(* CODESYS project Rasi_feeds_batching3.project

Project tree, tasks and I/O mapping:
  PLC_AC500_V3 : PM5032-T-ETH, ABB AG, order no. 1SAP123400R0x72, version 3.7.0.0
    application Application
      libraries: ModbusRtu, * (ABB); Util, * (System)
      task Task (cyclic, interval t#10ms, priority 14, watchdog t#20ms x 1) calls batching16
      CheckConfigurationObject
      Diagnosis/
        text list Diag_IO_Bus
        text list Diag_V3_PLC
      global variables GVL
      function block FB_Samyak_Multi [ST]
      function block FB_Samyak_Control [ST]
      function block Auto_Batching_V16 [ST]
      global variables PersistentVars
      function block Semi_Auto_Batching_V16 [ST]
      program batching16 [FBD]
    OnBoard_IO : 12DI/8DO-T/2DC, ABB AG, version 3.7.0.0
        input  E_Stop_DI : BOOL  // Fast inputs DI0-DI3.Digital input DI0
        input  Main_Cont_FB : BOOL  // Fast inputs DI0-DI3.Digital input DI1
        input  Auto_Mode_FB : BOOL  // Fast inputs DI0-DI3.Digital input DI2
        input  VFD_Run : BOOL  // Fast inputs DI0-DI3.Digital input DI3
        input  Start_PB : BOOL  // Fast inputs DI4-DI7.Digital input DI4
        output Auto_Bin1_Motor : BOOL  // Fast outputs DO0-DO3.Digital output DO0
        output Auto_Bin2_Motor : BOOL  // Fast outputs DO0-DO3.Digital output DO1
        output Auto_Bin3_Motor : BOOL  // Fast outputs DO0-DO3.Digital output DO2
        output Auto_Bin4_Motor : BOOL  // Fast outputs DO0-DO3.Digital output DO3
        output Auto_Bin5_Motor : BOOL  // Fast outputs DO4-DO7.Digital output DO4
        output Auto_Bin6_Motor : BOOL  // Fast outputs DO4-DO7.Digital output DO5
        output VFD_Slow : BOOL  // Fast outputs DO4-DO7.Digital output DO6
        unmapped channels: Fast inputs DI0-DI3, Fast inputs DI4-DI7, Standard inputs DI8-DI11, Digital inputs - Transistor, Fast outputs DO0-DO3, Fast outputs DO4-DO7, Digital outputs - Transistor
    IO_Bus : I/O-Bus, ABB AG, version 3.7.0.0
    Interfaces : Interfaces, ABB AG, version 3.7.0.0
      TA5142_RS485I : TA5142-RS485I, ABB AG, order no. 1SAP187300R0x02, version 3.7.0.0
        Modbus_RTU_Client : Modbus RTU Client, ABB AG, version 3.7.0.0
      OptionSlot_2
      Ethernet : Ethernet, ABB AG, version 3.7.0.0
        ETH1 : IP Settings, ABB AG, version 3.7.0.0
          NetConfig : NetConfig, ABB AG, version 3.7.0.0
          Modbus_TCP_IP_Server : Modbus TCP/IP Server, ABB AG, version 3.7.0.0
        Protocols : Client Protocols, ABB AG, version 3.7.0.0
    OnBoard_RTC : OnBoard RTC, ABB AG, version 3.7.0.0
  text list GlobalTextList
*)

// PLC_AC500_V3/Application/GVL
(* Part 1 of main GVL — HMI / %M tags only. Part 2: scripts/st_v16/GVL_RETAIN_PASTE.st *)
(* Combined: scripts/st_v16/GVL_LIVE_PLANT.st *)
{attribute 'qualified_only'}
VAR_GLOBAL
    Recipe_Weights AT %MD100: ARRAY [1..20] OF REAL;
	Semi_Auto_Bin_Material_Mapping AT %MW60: ARRAY [1..10] OF INT;	
	Auto_Bin_Material_Mapping AT %MW50: ARRAY[1..6] OF INT;	
	Auto_Coarse_To_Fine_speed AT %MD120: ARRAY[1..6] OF REAL := [1.0,1.0,1.0,1.0,1.0,1.0];
	Auto_Bin_Tolerance AT %MD150: ARRAY[1..6] OF REAL;
	Semi_Auto_Bin_Tolerance AT %MD160: ARRAY[1..10] OF REAL :=[0.2,0.2,0.2,0.2,0.2,0.2,0.2,0.2,0.2,0.2];
	Start_Button AT %MX2.0: BOOL;
	///E_Stop_Active AT %MX2.1: BOOL;
	Next_Cycle_Ready AT %MX2.2: BOOL;
	Reset AT %MX2.3: BOOL;
	Next_Cycle_Start AT %MX2.4: BOOL;
	Auto_Active_Mat AT %MW70: INT;
	Auto_Active_Bin AT %MW71: INT;
	Semi_Auto_Active_Mat AT %MW72: INT;
	Semi_Auto_Active_Bin AT %MW73: INT;
	Target_Batch_Cycles AT %MW74: INT := 0;
	Current_Batch_Cycle AT %MW75: INT;
	Completed_Batch_Cycles AT %MW79: INT;
	Error_Code AT %MW76: INT;
	Run AT %MX2.5 : BOOL;
	load_cell_auto AT %MD174 : REAL;
	load_cell_semi_auto AT %MD175 : REAL;
	Auto_Initial_Tolerance AT %MD176 : REAL := 5.0;
	Semi_Auto_Initial_Tolerance AT %MD178 : REAL := 5.0;
	Empty_Weight_Limit AT %MD186 : REAL := 5.0;
	Ex_Weight_Allow_kg AT %MD188 : REAL := 0.2;
	Auto_Total_Target_Weight AT %MD170 : REAL;
	Semi_Auto_Total_Target_Weight AT %MD171 : REAL;
	Auto_Total_Actual_Weight AT %MD180 : REAL;
	Semi_Auto_Total_Actual_Weight AT %MD184 : REAL;
	Auto_Material_Count AT %MW77: INT;
	Semi_Auto_Material_Count AT %MW78 : INT;
	Auto_Current_Step AT %MW80 : INT;
	Semi_Auto_Current_Step AT %MW81 : INT;
	Auto_Active_Target_Weight AT %MD220 : REAL;
	Semi_Auto_Active_Target_Weight AT %MD224 : REAL;
	Auto_Active_Live_Weight AT %MD172 : REAL;
	Semi_Auto_Active_Live_Weight AT %MD173 : REAL;
	Auto_Excess_Alarm AT %MX2.7 : BOOL;
	Semi_Auto_Excess_Alarm AT %MX2.8 : BOOL;
	Auto_Inter_Bin_Delay AT %MD190 : TIME;
	Semi_Auto_Inter_Bin_Delay AT %MD194 : TIME;
	Auto_Sequence_Complete AT %MX8.2 : BOOL;
	Semi_Auto_Sequence_Complete AT %MX8.3 : BOOL;
	All_Cycles_Complete AT %MX3.2 : BOOL;
	Auto_Status_Message : STRING(80);
	Semi_Auto_Status_Message : STRING(80);	
	Auto_Bin : ARRAY[1..6] OF BOOL;
	auto_motor_slow_trigger : ARRAY[1..6] OF BOOL;
	auto_bin_motor : ARRAY[1..6] OF BOOL;
	Semi_Auto_Bin : ARRAY[1..10] OF BOOL;
	Auto_Weights AT %MD300: ARRAY [1..6] OF REAL;
	Semi_Auto_Weights AT %MD350: ARRAY [1..10] OF REAL;
	Auto_Target_Weights AT %MD400: ARRAY [1..6] OF REAL;
	Semi_Auto_Target_Weights AT %MD410: ARRAY [1..10] OF REAL;
	Waiting_Next_batch_HMI_HIDE AT %MX8.1: BOOL;
	All_Cycles_Seq_Completed AT %MX8.4: BOOL;
	Done_Batch_HMI: BOOL;
	Error_bit AT %MX8.5: BOOL;
	Fault_Reset AT %MX8.6: BOOL;
	samyak_weight AT %MD195 : ARRAY[1..4] OF REAL;
	///samyak_weight_1: ARRAY[1..4] OF REAL;
END_VAR

// PLC_AC500_V3/Application/PersistentVars
VAR_GLOBAL PERSISTENT RETAIN
	(* HMI recipe/mapping shadow — no %M address; restored to GVL after power *)
	Ret_Recipe_Weights: ARRAY [1..20] OF REAL;
	bin_last_weight: REAL;
	Ret_Current_Step: INT;
	Ret_Cycle_Manager_State: INT;
	Ret_Internal_FB_Start: BOOL;
	Ret_bin_last_weight: REAL;
	Ret_GVL_Run: BOOL;
	Ret_Current_Batch_Cycle: INT;
	Ret_Completed_Batch_Cycles: INT;
	Ret_Target_Batch_Cycles: INT;
	Ret_Process_Was_Active: BOOL;
	Ret_Actual_Weights: ARRAY [1..6] OF REAL;
	Ret_Active_Material_ID: INT;
	Ret_Active_Bin_ID: INT;
	Ret_Active_Target_Weight: REAL;
	Ret_Active_Live_Weight: REAL;
	Ret_Resume_Step: INT;
	Ret_Bin_Target_Weights: ARRAY [1..6] OF REAL;
	Ret_Bin_Material_Mapping: ARRAY [1..6] OF INT;
	// Semi-Auto power resume (10 bins; steps 1..10 dosing, 31 settle, 32 complete)
	Ret_Semi_bin_last_weight: REAL;
	Ret_Semi_Current_Step: INT;
	Ret_Semi_Cycle_Manager_State: INT;
	Ret_Semi_Between_Cycle_Hold: BOOL;
	Ret_Semi_Last_Batch_Cycle: INT;
	Ret_Semi_GVL_Run: BOOL;
	Ret_Semi_Current_Batch_Cycle: INT;
	Ret_Semi_Completed_Batch_Cycles: INT;
	Ret_Semi_Target_Batch_Cycles: INT;
	Ret_Semi_Process_Was_Active: BOOL;
	Ret_Semi_Actual_Weights: ARRAY [1..10] OF REAL;
	Ret_Semi_Active_Material_ID: INT;
	Ret_Semi_Active_Bin_ID: INT;
	Ret_Semi_Active_Target_Weight: REAL;
	Ret_Semi_Active_Live_Weight: REAL;
	Ret_Semi_Resume_Step: INT;
	Ret_Semi_Bin_Target_Weights: ARRAY [1..10] OF REAL;
	Ret_Semi_Bin_Material_Mapping: ARRAY [1..10] OF INT;
END_VAR
VAR_GLOBAL PERSISTENT

END_VAR

// PLC_AC500_V3/Application/batching16
PROGRAM batching16
VAR
	Auto_Batching_V16_0: Auto_Batching_V16;
	Semi_Auto_Batching_V16_0: Semi_Auto_Batching_V16;
	FB_Samyak_Multi_2: FB_Samyak_Multi;
	arrTare_Cmds: ARRAY [1..4] OF BOOL;
	Auto_Msg: STRING(80);
	Semi_Auto_Err: INT;
	Semi_Auto_Msg: STRING(80);
END_VAR

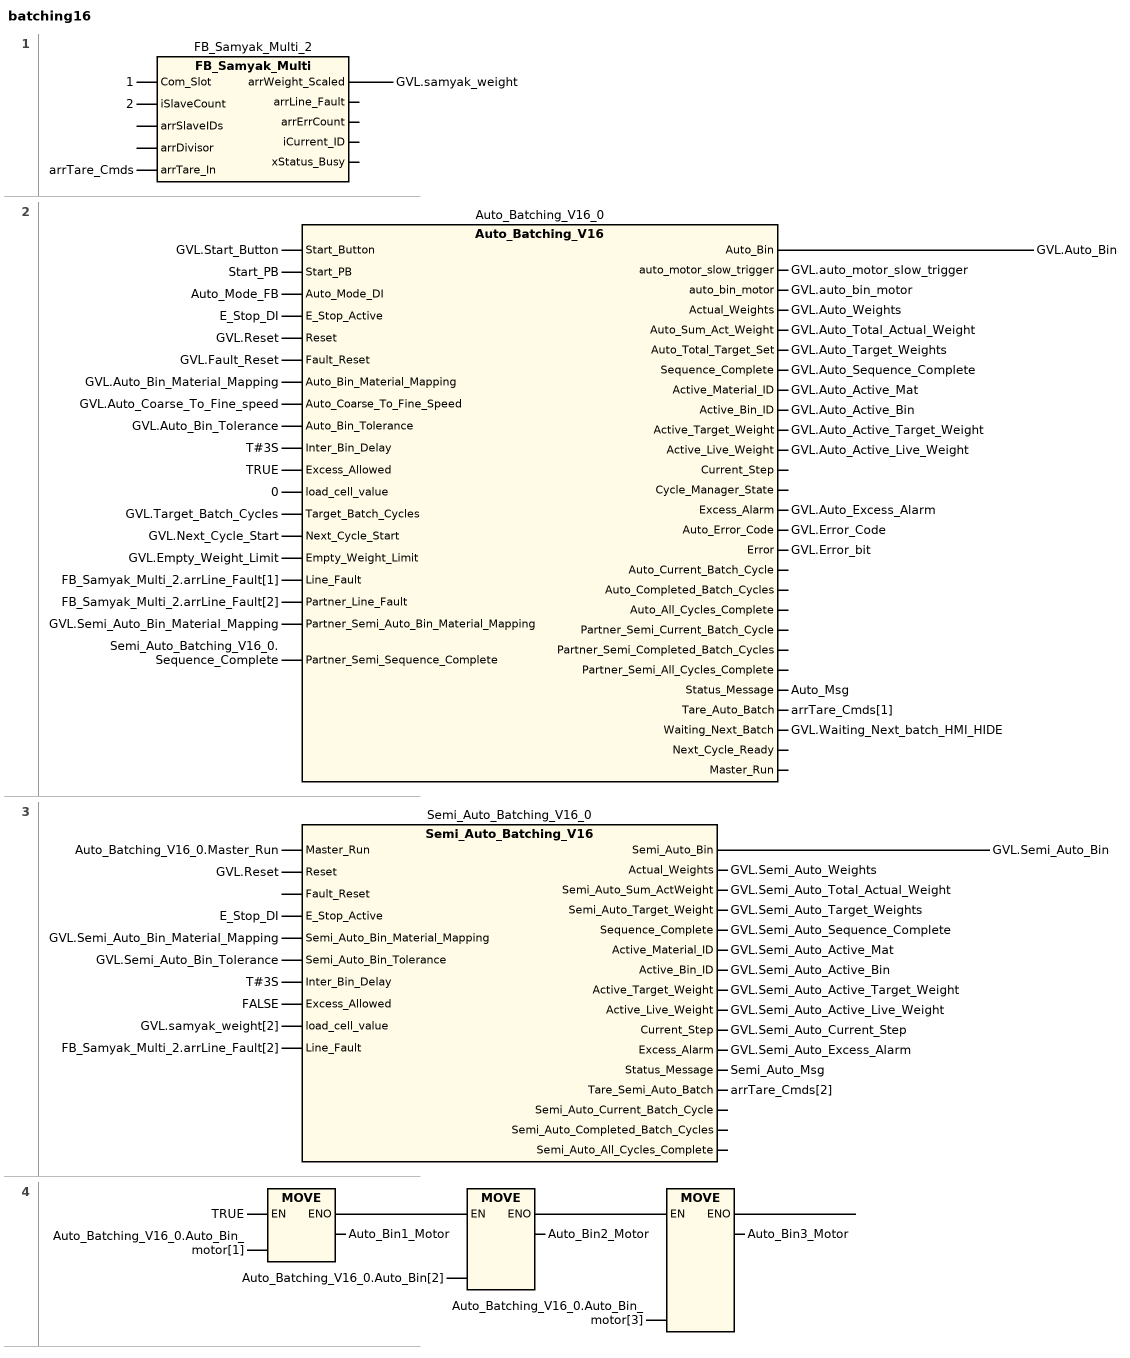
// NETWORK 1
FB_Samyak_Multi_2(Com_Slot := 1, iSlaveCount := 2, arrTare_In := arrTare_Cmds); // FB_Samyak_Multi
GVL.samyak_weight := FB_Samyak_Multi_2.arrWeight_Scaled;

// NETWORK 2
Auto_Batching_V16_0(
    Start_Button := GVL.Start_Button,
    Start_PB := Start_PB,
    Auto_Mode_DI := Auto_Mode_FB,
    E_Stop_Active := E_Stop_DI,
    Reset := GVL.Reset,
    Fault_Reset := GVL.Fault_Reset,
    Auto_Bin_Material_Mapping := GVL.Auto_Bin_Material_Mapping,
    Auto_Coarse_To_Fine_Speed := GVL.Auto_Coarse_To_Fine_speed,
    Auto_Bin_Tolerance := GVL.Auto_Bin_Tolerance,
    Inter_Bin_Delay := T#3S,
    Excess_Allowed := TRUE,
    load_cell_value := 0,
    Target_Batch_Cycles := GVL.Target_Batch_Cycles,
    Next_Cycle_Start := GVL.Next_Cycle_Start,
    Empty_Weight_Limit := GVL.Empty_Weight_Limit,
    Line_Fault := FB_Samyak_Multi_2.arrLine_Fault[1],
    Partner_Line_Fault := FB_Samyak_Multi_2.arrLine_Fault[2],
    Partner_Semi_Auto_Bin_Material_Mapping := GVL.Semi_Auto_Bin_Material_Mapping,
    Partner_Semi_Sequence_Complete := Semi_Auto_Batching_V16_0.Sequence_Complete,
    auto_motor_slow_trigger => GVL.auto_motor_slow_trigger,
    auto_bin_motor => GVL.auto_bin_motor,
    Actual_Weights => GVL.Auto_Weights,
    Auto_Sum_Act_Weight => GVL.Auto_Total_Actual_Weight,
    Auto_Total_Target_Set => GVL.Auto_Target_Weights,
    Sequence_Complete => GVL.Auto_Sequence_Complete,
    Active_Material_ID => GVL.Auto_Active_Mat,
    Active_Bin_ID => GVL.Auto_Active_Bin,
    Active_Target_Weight => GVL.Auto_Active_Target_Weight,
    Active_Live_Weight => GVL.Auto_Active_Live_Weight,
    Excess_Alarm => GVL.Auto_Excess_Alarm,
    Auto_Error_Code => GVL.Error_Code,
    Error => GVL.Error_bit,
    Status_Message => Auto_Msg,
    Tare_Auto_Batch => arrTare_Cmds[1],
    Waiting_Next_Batch => GVL.Waiting_Next_batch_HMI_HIDE); // Auto_Batching_V16
GVL.Auto_Bin := Auto_Batching_V16_0.Auto_Bin;

// NETWORK 3
Semi_Auto_Batching_V16_0(
    Master_Run := Auto_Batching_V16_0.Master_Run,
    Reset := GVL.Reset,
    E_Stop_Active := E_Stop_DI,
    Semi_Auto_Bin_Material_Mapping := GVL.Semi_Auto_Bin_Material_Mapping,
    Semi_Auto_Bin_Tolerance := GVL.Semi_Auto_Bin_Tolerance,
    Inter_Bin_Delay := T#3S,
    Excess_Allowed := FALSE,
    load_cell_value := GVL.samyak_weight[2],
    Line_Fault := FB_Samyak_Multi_2.arrLine_Fault[2],
    Actual_Weights => GVL.Semi_Auto_Weights,
    Semi_Auto_Sum_ActWeight => GVL.Semi_Auto_Total_Actual_Weight,
    Semi_Auto_Target_Weight => GVL.Semi_Auto_Target_Weights,
    Sequence_Complete => GVL.Semi_Auto_Sequence_Complete,
    Active_Material_ID => GVL.Semi_Auto_Active_Mat,
    Active_Bin_ID => GVL.Semi_Auto_Active_Bin,
    Active_Target_Weight => GVL.Semi_Auto_Active_Target_Weight,
    Active_Live_Weight => GVL.Semi_Auto_Active_Live_Weight,
    Current_Step => GVL.Semi_Auto_Current_Step,
    Excess_Alarm => GVL.Semi_Auto_Excess_Alarm,
    Status_Message => Semi_Auto_Msg,
    Tare_Semi_Auto_Batch => arrTare_Cmds[2]); // Semi_Auto_Batching_V16
GVL.Semi_Auto_Bin := Semi_Auto_Batching_V16_0.Semi_Auto_Bin;

// NETWORK 4
Auto_Bin1_Motor := Auto_Batching_V16_0.Auto_Bin_motor[1];
Auto_Bin2_Motor := Auto_Batching_V16_0.Auto_Bin[2];
Auto_Bin3_Motor := Auto_Batching_V16_0.Auto_Bin_motor[3];

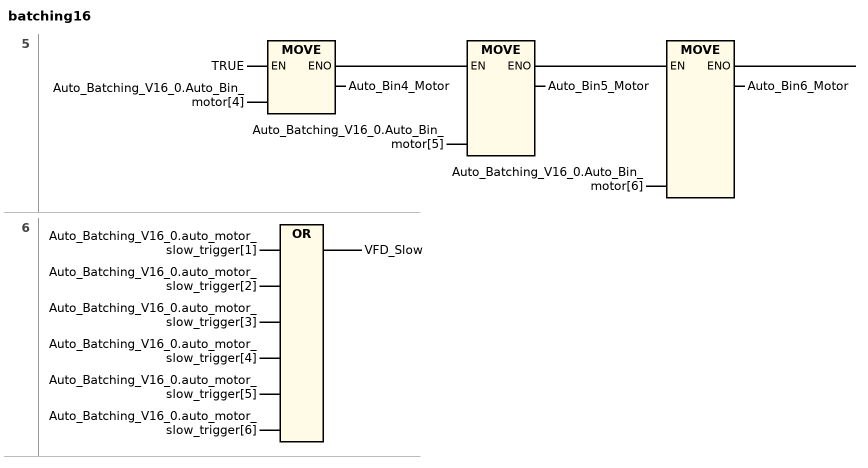
// NETWORK 5
Auto_Bin4_Motor := Auto_Batching_V16_0.Auto_Bin_motor[4];
Auto_Bin5_Motor := Auto_Batching_V16_0.Auto_Bin_motor[5];
Auto_Bin6_Motor := Auto_Batching_V16_0.Auto_Bin_motor[6];

// NETWORK 6
VFD_Slow := Auto_Batching_V16_0.auto_motor_slow_trigger[1] OR Auto_Batching_V16_0.auto_motor_slow_trigger[2] OR Auto_Batching_V16_0.auto_motor_slow_trigger[3] OR Auto_Batching_V16_0.auto_motor_slow_trigger[4] OR Auto_Batching_V16_0.auto_motor_slow_trigger[5] OR Auto_Batching_V16_0.auto_motor_slow_trigger[6];

END_PROGRAM

// PLC_AC500_V3/Application/FB_Samyak_Multi
//SAMYAK 4016 Multi Slave Unit Customised Block
//Note: This FB_Samyak_Multi name is impotrtant when you create new POU.

FUNCTION_BLOCK FB_Samyak_Multi
VAR_INPUT
    Com_Slot      : BYTE := 1;    (* Port Number *)
    iSlaveCount   : INT := 1;     (* How many slaves active: 1 to 4 *)
    arrSlaveIDs   : ARRAY[1..4] OF BYTE := [1, 2, 3, 4]; (* Unit IDs *)
    // Scaling per Unit
	arrDivisor: ARRAY [1..4] OF REAL := [10.0, 10.0, 10.0, 10.0];
    arrTare_In    : ARRAY[1..4] OF BOOL; (* Individual Tare triggers *)
END_VAR

VAR_OUTPUT
    arrWeight_Scaled : ARRAY[1..4] OF REAL; (* Scaled result per unit *)
    arrLine_Fault    : ARRAY[1..4] OF BOOL; (* Fault status per unit *)
    arrErrCount      : ARRAY[1..4] OF INT;  (* Error count per unit *)
    iCurrent_ID      : BYTE;                (* Current ID being polled *)
    xStatus_Busy     : BOOL;                (* Overall Bus Busy *)
END_VAR

VAR
    (* Internal ModRtuMast Instances *)
    fbRead         : ModRtuMast;
    fbTare         : ModRtuMast;
    
    (* Polling Control *)
    iStep          : INT := 0;
    iIdx           : INT := 1;    (* Current Loop Index *)
    Samyak_Buffer  : ARRAY[0..17] OF WORD;
    wTareCommand   : WORD := 1;
    
    (* Unique Timer/Trigger Instances *)
    rtTareTrig     : R_TRIG;
    rtErrTrig      : R_TRIG;
    tWatchdog      : TON;
    tRecovery      : TON;
END_VAR



(* --- 1. INDIVIDUAL UNIT MONITORING --- *)
iCurrent_ID := arrSlaveIDs[iIdx]; 

(* Watchdog for Bus Hangs *)
tWatchdog(IN := (fbRead.Busy OR fbTare.Busy), PT := T#2000MS);
xStatus_Busy := fbRead.Busy OR fbTare.Busy;

(* Error Tracking for Current Index *)
rtErrTrig(CLK := (fbRead.Error OR fbTare.Error));
IF rtErrTrig.Q THEN
    arrErrCount[iIdx] := arrErrCount[iIdx] + 1;
END_IF

(* Reset on Success *)
IF fbRead.Done OR fbTare.Done THEN
    arrErrCount[iIdx] := 0;
    arrLine_Fault[iIdx] := FALSE;
END_IF

(* Line Fault Activation (10 errors) *)
IF arrErrCount[iIdx] >= 10 THEN
    arrLine_Fault[iIdx] := TRUE;
END_IF

(* Auto-Recovery pulse (5s) *)
tRecovery(IN := arrLine_Fault[iIdx], PT := T#5S);
IF tRecovery.Q THEN
    arrErrCount[iIdx] := 0;
    arrLine_Fault[iIdx] := FALSE;
END_IF

IF tWatchdog.Q THEN iStep := 99; END_IF

(* Check Tare for active slave *)
rtTareTrig(CLK := arrTare_In[iIdx]);

(* --- 2. SEQUENTIAL STATE MACHINE --- *)
CASE iStep OF
    
    0: (* READ CURRENT SLAVE *)
        fbTare(Execute := FALSE);
        fbRead(
            Execute := NOT (fbRead.Done OR fbRead.Error OR fbRead.Busy) 
                       AND NOT rtTareTrig.Q AND NOT arrLine_Fault[iIdx],
            COM     := Com_Slot,
            Serv    := arrSlaveIDs[iIdx],
            FCT     := 3, Addr := 0, Nb := 2, 
            Data    := ADR(Samyak_Buffer[0]), Timeout := 400
        );

        IF fbRead.Done THEN
            (* Scale weight using the array-based divisor for this specific index *)
            arrWeight_Scaled[iIdx] := TO_REAL(TO_DINT(SHL(TO_DWORD(Samyak_Buffer[1]), 16) OR TO_DWORD(Samyak_Buffer[0]))) / arrDivisor[iIdx];
            iStep := 10; (* Switch to next slave *)
        END_IF
        
        IF fbRead.Error THEN iStep := 10; END_IF (* Move on if error *)
        IF rtTareTrig.Q THEN iStep := 1; END_IF  (* Priority: Tare current unit *)

    1: (* PORT RELEASE *)
        fbRead(Execute := FALSE);
        IF NOT fbRead.Busy THEN iStep := 2; END_IF

    2: (* WRITE TARE FOR CURRENT SLAVE *)
        fbTare(
            Execute := TRUE,
            COM := Com_Slot, Serv := arrSlaveIDs[iIdx], 
            FCT := 6, Addr := 16, Nb := 1,
            Data := ADR(wTareCommand), Timeout := 1000
        );

        IF fbTare.Done OR fbTare.Error THEN
            arrTare_In[iIdx] := FALSE; (* Reset manual trigger *)
            iStep := 3;
        END_IF

    3: (* CLEANUP *)
        fbTare(Execute := FALSE);
        IF NOT fbTare.Busy THEN iStep := 10; END_IF

    10: (* INDEX ROTATION *)
        iIdx := iIdx + 1;
        IF iIdx > iSlaveCount THEN
            iIdx := 1; (* Back to first slave *)
        END_IF
        iStep := 0;

    99: (* EMERGENCY RESET *)
        fbRead(Execute := FALSE); fbTare(Execute := FALSE);
        IF NOT (fbRead.Busy OR fbTare.Busy) THEN iStep := 0; END_IF
        
END_CASE

END_FUNCTION_BLOCK

// PLC_AC500_V3/Application/Auto_Batching_V16
FUNCTION_BLOCK Auto_Batching_V16
VAR_INPUT
    Start_Button : BOOL;                            // Master start command from HMI (%MX2.0)
    Start_PB : BOOL;                                // Physical Start pushbutton DI (one-shot pulse)
    Auto_Mode_DI : BOOL;                            // Auto Mode DI: TRUE = process start allowed; FALSE = HMI/PB start ignored
    E_Stop_Active : BOOL;                           // Emergency Stop circuit status (NC contact: TRUE = Healthy/Run permitted, FALSE = E-Stop tripped)
    Reset : BOOL;                                   // Production abort: clears steps, weights, cycles, CMS.
    Fault_Reset : BOOL;                             // Rising-edge fault acknowledge: clears Error_Code if live fault cleared
    Auto_Bin_Material_Mapping : ARRAY[1..6] OF INT; // Array mapping physical Silos 1..6 to Recipe Material IDs (1..20, 0 = Silo skipped)
    Auto_Coarse_To_Fine_Speed : ARRAY[1..6] OF REAL;// Weight offset threshold (kg) before target to transition from Coarse to Fine feeding
    Auto_Bin_Tolerance : ARRAY[1..6] OF REAL;       // Allowable weight tolerance window (±kg) around target weight for each silo
    Inter_Bin_Delay : TIME := T#5S;                 // Pause after Bin*=FALSE: tailings on SAME bin ID; then next mat (Auto e.g. T#5S)
    Excess_Allowed : BOOL := FALSE;                 // Overfill handling policy: TRUE = proceed if target is exceeded, FALSE = raise alarm and halt
    load_cell_value : REAL;                         // Live gross weight input reading from the Auto scale load cell (kg)
    Target_Batch_Cycles : INT := 1;                 // Target number of batch cycle repetitions configured from HMI (defaults to 1)
    Next_Cycle_Start : BOOL;                        // NextBatchStart: after a completed cycle (Target>1), press when this FB scale < Empty_Weight_Limit
    Empty_Weight_Limit : REAL := 0.5;               // Both scales must be LT this (kg) before Start/Start_PB, Next_Cycle_Start, or Tare pulse
    Line_Fault : BOOL;                              // Auto scale arrLine_Fault. TRUE => Auto_Error_Code=5 + HOLD
    Partner_Line_Fault : BOOL;                      // Partner Semi load-cell comms fail (arrLine_Fault). TRUE => Auto_Error_Code=8
    Partner_Semi_Auto_Bin_Material_Mapping : ARRAY[1..10] OF INT; // Semi silo Mat IDs 1..10 (wire GVL.Semi_Auto_Bin_Material_Mapping)
    Partner_Semi_Sequence_Complete : BOOL;          // Handshake input from Follower (Semi-Auto) Sequence_Complete
END_VAR
VAR_OUTPUT
    Auto_Bin : ARRAY[1..6] OF BOOL;                 // Coarse feeding valve / gate actuation command outputs for Silos 1..6
    auto_motor_slow_trigger : ARRAY[1..6] OF BOOL;  // Fine feeding valve / VFD slow speed command outputs for Silos 1..6
    auto_bin_motor : ARRAY[1..6] OF BOOL;           // Feeder / screw conveyor motor run commands for Silos 1..6
    Actual_Weights : ARRAY[1..6] OF REAL;           // Net material weight (kg) successfully dosed for each silo in the current cycle
    Auto_Sum_Act_Weight : REAL;                     // Sum of Actual_Weights[1..6]
    Auto_Total_Target_Set : ARRAY[1..6] OF REAL;    // Per-bin target kg (bin index 1..6)
    Sequence_Complete : BOOL;                       // Auto Sequence Complete (Step 8 reached)
    Active_Material_ID : INT;                       // Recipe Material ID currently being dosed (1..20, 0 when idle/complete)
    Active_Bin_ID : INT;                            // Physical Silo index currently being dosed (1..6, 0 when idle/complete)
    Active_Target_Weight : REAL;                    // Target weight setpoint (kg) of the ingredient currently being dosed
    Active_Live_Weight : REAL;                      // Live net/tared weight (kg) accumulated into the scale for the active silo
    Current_Step : INT;                             // Real-time sequence step: 0=Idle, 1..6=Dosing, 7=Settle, 8=Complete
    Cycle_Manager_State : INT;                      // Master supervisory state: 0=Idle, 1=Running, 4=All Done, 5=Between Cycles Hold
    Excess_Alarm : BOOL;                            // Overfill alarm
    
    (* =========================================================================
       MASTER SYSTEM ERROR CODES REFERENCE (Displayed in GVL.Error_Code %MW76):
       0  = System Healthy / No Error
       1  = Auto Duplicate Material ID (within Silos 1..6)
       2  = Auto Invalid Material ID (< 0 or > 20)
       3  = Auto Target Weight < (Coarse_To_Fine_Speed + Tolerance)
       4  = Auto Scale 1 Not Empty (> Empty_Weight_Limit) at Start / Cycle Trigger
       5  = Auto Scale 1 Communication Line Fault (FB_Samyak_Multi Scale 1)
       6  = Recipe / Bin Mapping is all 0s (no ingredients assigned)
       7  = Cross-Scale Duplicate Material (Same Material mapped on Auto and Semi)
       8  = Semi Scale 2 Communication Line Fault (FB_Samyak_Multi Scale 2)
       9  = Semi Duplicate Material ID (within Silos 1..10)
       10 = Semi Scale 2 Not Empty (> Empty_Weight_Limit) at Start / Cycle Trigger
       11 = Semi Invalid Material ID (< 0 or > 20)
       12 = Semi Target Weight < (Coarse_To_Fine_Speed + Tolerance)
       ========================================================================= *)
    Auto_Error_Code : INT;                          // Fault diagnostic code (0=OK, 1..12)
    Error : BOOL;                                   // TRUE when Auto_Error_Code > 0
    Auto_Current_Batch_Cycle : INT;                 // Active batch cycle number currently processing (1..Target_Batch_Cycles)
    Auto_Completed_Batch_Cycles : INT;              // Total number of batch cycle loops completed successfully
    Auto_All_Cycles_Complete : BOOL;                // Master flag: TRUE when all Target_Batch_Cycles have finished
    Partner_Semi_Current_Batch_Cycle : INT;         // Follower (Semi) cycle number mirroring GVL
    Partner_Semi_Completed_Batch_Cycles : INT;      // Follower (Semi) completed cycles
    Partner_Semi_All_Cycles_Complete : BOOL;        // Follower (Semi) all cycles complete flag
    Status_Message : STRING(80);                    // Diagnostic status message
    Tare_Auto_Batch : BOOL;                         // One-scan pulse to Auto scale load cell indicator
    Waiting_Next_Batch : BOOL;                      // TRUE in State 5 between cycles
    Next_Cycle_Ready : BOOL;                        // TRUE when both scales are confirmed empty and debounced in State 5
    
    // Master-to-Follower Single Coordination Signal
    Master_Run : BOOL;                              // Master Run signal wired directly to Semi-Auto Follower
END_VAR
VAR
    bin_last_weight : REAL;
    actual_bin : REAL;
    target_weight : REAL;
    cutoff_trigger_weight : REAL;
    min_tol_weight : REAL;
    max_tol_weight : REAL;
    Paused_By_Hold : BOOL;
    Effective_Delay : TIME;
    Inter_Bin_Settling : BOOL;
    Inter_Bin_Settle_Arm : INT;
    Inter_Bin_Timer : TON;
    Periodic_Check_Timer : TON;
    Settle_Hold_Step : INT;
    Settle_Hold_Mat : INT;
    Settle_Hold_Target : REAL;
    Inter_Bin_Next_Step : INT;
    Mat_Idx : INT;
    j_Mat : INT;
    i : INT;
    j : INT;
    Completion_Timer : TON;
    Empty_Debounce_Timer : TON;                     // 1s debounce filter for empty scale verification in State 5
    Internal_FB_Start : BOOL;
    Duplicate_Found : BOOL;
    Duplicate_Vs_Partner : BOOL;
    Duplicate_Partner_Internal : BOOL;
    Auto_Mapping_All_Zero : BOOL;
    Partner_Mapping_All_Zero : BOOL;
    Invalid_Material_Range : BOOL;
    Weight_Limit_Error : BOOL;
    Semi_Invalid_Material_Range : BOOL;
    Semi_Weight_Limit_Error : BOOL;
    eff_empty_limit : REAL;
    Scale_Empty_OK : BOOL;
    Next_Cycle_Last : BOOL;
    Next_Cycle_Rising : BOOL;
    Tare_Pulse_Req : BOOL;
    Start_Cmd : BOOL;
    Start_Cmd_Last : BOOL;
    Start_Pulse : BOOL;
    First_Scan_Done : BOOL;
    Auto_Has_Active_Bins : BOOL;
    Semi_Has_Active_Bins : BOOL;
    Reset_Last : BOOL;
    Reset_Pulse : BOOL;
    Fault_Reset_Last : BOOL;
    Fault_Reset_Pulse : BOOL;
    Between_Cycle_Hold : BOOL;
    Last_Dosing_Step : INT;
    Semi_Sequence_Done : BOOL;
END_VAR

// -----------------------------------------------------------------------------
// 0. TIMINGS, THRESHOLDS & EDGE DETECTION
// -----------------------------------------------------------------------------
Effective_Delay := Inter_Bin_Delay;
IF Effective_Delay = T#0S THEN
    Effective_Delay := T#2S;
END_IF;

eff_empty_limit := Empty_Weight_Limit;
IF eff_empty_limit <= 0.0 THEN
    eff_empty_limit := GVL.Empty_Weight_Limit;
END_IF;
IF eff_empty_limit <= 0.0 THEN
    eff_empty_limit := 0.5;
END_IF;

Scale_Empty_OK := (load_cell_value < eff_empty_limit) AND (GVL.load_cell_auto < eff_empty_limit)
    AND (GVL.load_cell_semi_auto < eff_empty_limit);

Start_Cmd := (Start_Button OR GVL.Start_Button OR Start_PB) AND Auto_Mode_DI;
Start_Pulse := Start_Cmd AND NOT Start_Cmd_Last;
Start_Cmd_Last := Start_Cmd;

Next_Cycle_Rising := (Next_Cycle_Start OR GVL.Next_Cycle_Start) AND NOT Next_Cycle_Last;
Next_Cycle_Last := (Next_Cycle_Start OR GVL.Next_Cycle_Start);

Reset_Pulse := (Reset OR GVL.Reset) AND NOT Reset_Last;
Reset_Last := (Reset OR GVL.Reset);

Fault_Reset_Pulse := Fault_Reset AND NOT Fault_Reset_Last;
Fault_Reset_Last := Fault_Reset;

// Combine direct pin and GVL handshake for Follower completion
Semi_Sequence_Done := Partner_Semi_Sequence_Complete OR GVL.Semi_Auto_Sequence_Complete;

// -----------------------------------------------------------------------------
// 1. FIRST SCAN POWER-RESUME & RETAIN RESTORE
// -----------------------------------------------------------------------------
IF NOT First_Scan_Done THEN
    First_Scan_Done := TRUE;
    
    // Restore HMI Recipe & Mapping retain if GVL uninitialized
    FOR i := 1 TO 20 DO
        IF (GVL.Recipe_Weights[i] <= 0.001) AND (PersistentVars.Ret_Recipe_Weights[i] > 0.001) THEN
            GVL.Recipe_Weights[i] := PersistentVars.Ret_Recipe_Weights[i];
        END_IF;
    END_FOR;
    FOR i := 1 TO 6 DO
        IF (GVL.Auto_Bin_Material_Mapping[i] = 0) AND (PersistentVars.Ret_Bin_Material_Mapping[i] > 0) THEN
            GVL.Auto_Bin_Material_Mapping[i] := PersistentVars.Ret_Bin_Material_Mapping[i];
        END_IF;
    END_FOR;
    FOR i := 1 TO 10 DO
        IF (GVL.Semi_Auto_Bin_Material_Mapping[i] = 0) AND (PersistentVars.Ret_Semi_Bin_Material_Mapping[i] > 0) THEN
            GVL.Semi_Auto_Bin_Material_Mapping[i] := PersistentVars.Ret_Semi_Bin_Material_Mapping[i];
        END_IF;
    END_FOR;

    // Power Resume: restore exact state without corrupting actual weights with live load cell
    IF PersistentVars.Ret_Process_Was_Active AND (PersistentVars.Ret_Cycle_Manager_State = 1) 
       AND (PersistentVars.Ret_Resume_Step >= 1) AND (PersistentVars.Ret_Resume_Step <= 6) THEN
        
        Current_Step := PersistentVars.Ret_Resume_Step;
        Last_Dosing_Step := Current_Step;
        Cycle_Manager_State := 1;
        Internal_FB_Start := TRUE;
        Between_Cycle_Hold := FALSE;
        GVL.Run := TRUE;
        Master_Run := TRUE;
        GVL.Current_Batch_Cycle := PersistentVars.Ret_Current_Batch_Cycle;
        GVL.Completed_Batch_Cycles := PersistentVars.Ret_Completed_Batch_Cycles;
        IF PersistentVars.Ret_Target_Batch_Cycles > 0 THEN
            GVL.Target_Batch_Cycles := PersistentVars.Ret_Target_Batch_Cycles;
        END_IF;

        bin_last_weight := PersistentVars.Ret_bin_last_weight;
        PersistentVars.bin_last_weight := bin_last_weight;

        // Reconcile with live load cell weight to account for extra material dumped while power was off
        IF (load_cell_value >= bin_last_weight) AND NOT Line_Fault THEN
            Active_Live_Weight := load_cell_value - bin_last_weight;
            Actual_Weights[Current_Step] := Active_Live_Weight;
        ELSE
            Active_Live_Weight := PersistentVars.Ret_Active_Live_Weight;
            Actual_Weights[Current_Step] := Active_Live_Weight;
        END_IF;

        Auto_Sum_Act_Weight := 0.0;
        FOR i := 1 TO 6 DO
            IF i <> Current_Step THEN
                Actual_Weights[i] := PersistentVars.Ret_Actual_Weights[i];
            END_IF;
            GVL.Auto_Weights[i] := Actual_Weights[i];
            Auto_Sum_Act_Weight := Auto_Sum_Act_Weight + Actual_Weights[i];
        END_FOR;
        GVL.Auto_Total_Actual_Weight := Auto_Sum_Act_Weight;

        GVL.Auto_Active_Live_Weight := Active_Live_Weight;
        Active_Material_ID := PersistentVars.Ret_Active_Material_ID;
        Active_Bin_ID := PersistentVars.Ret_Active_Bin_ID;
        Active_Target_Weight := PersistentVars.Ret_Active_Target_Weight;
        GVL.Auto_Active_Mat := Active_Material_ID;
        GVL.Auto_Active_Bin := Active_Bin_ID;
        GVL.Auto_Active_Target_Weight := Active_Target_Weight;

        Paused_By_Hold := TRUE;
        Tare_Pulse_Req := FALSE;
        Tare_Auto_Batch := FALSE;

        // Check if material dumped during power-off has already reached or exceeded target weight
        IF (Active_Target_Weight > 0.0) AND (Active_Live_Weight >= (Active_Target_Weight - Auto_Bin_Tolerance[Current_Step])) THEN
            IF Active_Live_Weight > (Active_Target_Weight + Auto_Bin_Tolerance[Current_Step]) THEN
                Status_Message := CONCAT('Auto [POWER RESUME]: Step ', CONCAT(INT_TO_STRING(Current_Step), ' Overfilled — Waiting Resume'));
            ELSE
                Status_Message := CONCAT('Auto [POWER RESUME]: Step ', CONCAT(INT_TO_STRING(Current_Step), ' Target Reached — Advancing on Resume'));
            END_IF;
        ELSE
            Status_Message := CONCAT('Auto [POWER RESUME]: Step ', CONCAT(INT_TO_STRING(Current_Step), ' Resumed — Ready to Feed'));
        END_IF;

    ELSIF (PersistentVars.Ret_Cycle_Manager_State = 5) THEN
        Cycle_Manager_State := 5;
        Between_Cycle_Hold := TRUE;
        Current_Step := 8;
        Sequence_Complete := TRUE;
        GVL.Auto_Sequence_Complete := TRUE;
        GVL.Run := TRUE;
        Master_Run := TRUE;
        GVL.Current_Batch_Cycle := PersistentVars.Ret_Current_Batch_Cycle;
        GVL.Completed_Batch_Cycles := PersistentVars.Ret_Completed_Batch_Cycles;
        IF PersistentVars.Ret_Target_Batch_Cycles > 0 THEN
            GVL.Target_Batch_Cycles := PersistentVars.Ret_Target_Batch_Cycles;
        END_IF;
        FOR i := 1 TO 6 DO
            Actual_Weights[i] := PersistentVars.Ret_Actual_Weights[i];
            GVL.Auto_Weights[i] := Actual_Weights[i];
        END_FOR;
        Tare_Pulse_Req := FALSE;
        Tare_Auto_Batch := FALSE;
        Status_Message := 'Auto [POWER RESUME]: State 5 - Waiting empty scale & Next_Cycle_Start';

    ELSE
        Current_Step := 0;
        Cycle_Manager_State := 0;
        Internal_FB_Start := FALSE;
        Master_Run := FALSE;
        Between_Cycle_Hold := FALSE;
        Sequence_Complete := FALSE;
        Tare_Pulse_Req := FALSE;
        Tare_Auto_Batch := FALSE;
        Next_Cycle_Ready := FALSE;
        Status_Message := 'Auto [Idle]: Ready - Waiting for Start';
    END_IF;
END_IF;

// Retain snapshot of HMI mappings
FOR i := 1 TO 20 DO
    PersistentVars.Ret_Recipe_Weights[i] := GVL.Recipe_Weights[i];
END_FOR;
FOR i := 1 TO 6 DO
    PersistentVars.Ret_Bin_Material_Mapping[i] := GVL.Auto_Bin_Material_Mapping[i];
END_FOR;
FOR i := 1 TO 10 DO
    PersistentVars.Ret_Semi_Bin_Material_Mapping[i] := GVL.Semi_Auto_Bin_Material_Mapping[i];
END_FOR;

// -----------------------------------------------------------------------------
// 2. CONFIGURATION CHECKS & ERROR DIAGNOSTICS
// -----------------------------------------------------------------------------
Duplicate_Found := FALSE;
Duplicate_Vs_Partner := FALSE;
Duplicate_Partner_Internal := FALSE;
Auto_Mapping_All_Zero := TRUE;
Partner_Mapping_All_Zero := TRUE;
Invalid_Material_Range := FALSE;
Weight_Limit_Error := FALSE;
Auto_Has_Active_Bins := FALSE;
Semi_Has_Active_Bins := FALSE;

GVL.Auto_Total_Target_Weight := 0.0;
GVL.Auto_Material_Count := 0;

FOR i := 1 TO 6 DO
    Mat_Idx := Auto_Bin_Material_Mapping[i];
    IF (Mat_Idx < 1) OR (Mat_Idx > 20) THEN
        Mat_Idx := GVL.Auto_Bin_Material_Mapping[i];
    END_IF;
    IF Mat_Idx <> 0 THEN
        Auto_Mapping_All_Zero := FALSE;
    END_IF;
    IF (Mat_Idx < 0) OR (Mat_Idx > 20) THEN
        Invalid_Material_Range := TRUE;
    END_IF;
    IF (Mat_Idx >= 1) AND (Mat_Idx <= 20) THEN
        FOR j := 1 TO 6 DO
            IF j <> i THEN
                j_Mat := Auto_Bin_Material_Mapping[j];
                IF (j_Mat < 1) OR (j_Mat > 20) THEN
                    j_Mat := GVL.Auto_Bin_Material_Mapping[j];
                END_IF;
                IF (j_Mat = Mat_Idx) THEN
                    Duplicate_Found := TRUE;
                END_IF;
            END_IF;
        END_FOR;
        FOR j := 1 TO 10 DO
            j_Mat := Partner_Semi_Auto_Bin_Material_Mapping[j];
            IF (j_Mat < 1) OR (j_Mat > 20) THEN
                j_Mat := GVL.Semi_Auto_Bin_Material_Mapping[j];
            END_IF;
            IF (j_Mat = Mat_Idx) THEN
                Duplicate_Vs_Partner := TRUE;
            END_IF;
        END_FOR;
        target_weight := GVL.Recipe_Weights[Mat_Idx];
        IF target_weight > 0.0 THEN
            GVL.Auto_Total_Target_Weight := GVL.Auto_Total_Target_Weight + target_weight;
            GVL.Auto_Material_Count := GVL.Auto_Material_Count + 1;
            Auto_Has_Active_Bins := TRUE;
            IF target_weight < (Auto_Coarse_To_Fine_Speed[i] + Auto_Bin_Tolerance[i]) THEN
                Weight_Limit_Error := TRUE;
            END_IF;
        END_IF;
    END_IF;
END_FOR;

Semi_Invalid_Material_Range := FALSE;
Semi_Weight_Limit_Error := FALSE;

FOR i := 1 TO 10 DO
    Mat_Idx := Partner_Semi_Auto_Bin_Material_Mapping[i];
    IF (Mat_Idx < 1) OR (Mat_Idx > 20) THEN
        Mat_Idx := GVL.Semi_Auto_Bin_Material_Mapping[i];
    END_IF;
    IF Mat_Idx <> 0 THEN
        Partner_Mapping_All_Zero := FALSE;
    END_IF;
    IF (Mat_Idx < 0) OR (Mat_Idx > 20) THEN
        Semi_Invalid_Material_Range := TRUE;
    END_IF;
    IF (Mat_Idx >= 1) AND (Mat_Idx <= 20) THEN
        FOR j := 1 TO 10 DO
            IF j <> i THEN
                j_Mat := Partner_Semi_Auto_Bin_Material_Mapping[j];
                IF (j_Mat < 1) OR (j_Mat > 20) THEN
                    j_Mat := GVL.Semi_Auto_Bin_Material_Mapping[j];
                END_IF;
                IF (j_Mat = Mat_Idx) THEN
                    Duplicate_Partner_Internal := TRUE;
                END_IF;
            END_IF;
        END_FOR;
        target_weight := GVL.Recipe_Weights[Mat_Idx];
        IF target_weight > 0.0 THEN
            Semi_Has_Active_Bins := TRUE;
            IF target_weight < GVL.Semi_Auto_Bin_Tolerance[i] THEN
                Semi_Weight_Limit_Error := TRUE;
            END_IF;
        END_IF;
    END_IF;
END_FOR;

IF Line_Fault THEN
    Auto_Error_Code := 5;
    GVL.Error_Code := 5;
    Status_Message := 'Auto_Error_Code 5: Auto Scale 1 Line_Fault Error!';
ELSIF Partner_Line_Fault THEN
    Auto_Error_Code := 8;
    GVL.Error_Code := 8;
    Status_Message := 'Auto_Error_Code 8: Semi Scale 2 Line_Fault Error!';
ELSIF Auto_Mapping_All_Zero AND Partner_Mapping_All_Zero THEN
    Auto_Error_Code := 6;
    GVL.Error_Code := 6;
    Status_Message := 'Auto_Error_Code 6: Mapping is all 0!';
ELSIF Duplicate_Found THEN
    Auto_Error_Code := 1;
    GVL.Error_Code := 1;
    Status_Message := 'Auto_Error_Code 1: Duplicate Material ID within Auto bins!';
ELSIF Duplicate_Partner_Internal THEN
    Auto_Error_Code := 9;
    GVL.Error_Code := 9;
    Status_Message := 'Auto_Error_Code 9: Duplicate Material ID inside Semi mapping!';
ELSIF Duplicate_Vs_Partner THEN
    Auto_Error_Code := 7;
    GVL.Error_Code := 7;
    Status_Message := 'Auto_Error_Code 7: Material ID duplicated on Auto and Semi!';
ELSIF Invalid_Material_Range THEN
    Auto_Error_Code := 2;
    GVL.Error_Code := 2;
    Status_Message := 'Auto_Error_Code 2: Auto Material Index out of range (1..20)!';
ELSIF Semi_Invalid_Material_Range THEN
    Auto_Error_Code := 11;
    GVL.Error_Code := 11;
    Status_Message := 'Auto_Error_Code 11: Semi Material Index out of range (1..20)!';
ELSIF Weight_Limit_Error THEN
    Auto_Error_Code := 3;
    GVL.Error_Code := 3;
    Status_Message := 'Auto_Error_Code 3: Auto Recipe weight < Coarse_To_Fine + Tolerance!';
ELSIF Semi_Weight_Limit_Error THEN
    Auto_Error_Code := 12;
    GVL.Error_Code := 12;
    Status_Message := 'Auto_Error_Code 12: Semi Recipe weight < Tolerance!';
ELSIF (Auto_Error_Code <> 4) AND (Auto_Error_Code <> 10) THEN
    Auto_Error_Code := 0;
    IF (GVL.Error_Code <> 4) AND (GVL.Error_Code <> 10) THEN
        GVL.Error_Code := 0;
    END_IF;
END_IF;

Error := (Auto_Error_Code > 0);

// -----------------------------------------------------------------------------
// 3. MASTER RESET & FAULT RESET
// -----------------------------------------------------------------------------
IF Reset_Pulse THEN
    FOR i := 1 TO 6 DO
        Auto_Bin[i] := FALSE;
        auto_motor_slow_trigger[i] := FALSE;
        auto_bin_motor[i] := FALSE;
        Actual_Weights[i] := 0.0;
        Auto_Total_Target_Set[i] := 0.0;
        GVL.Auto_Bin[i] := FALSE;
        GVL.auto_motor_slow_trigger[i] := FALSE;
        GVL.auto_bin_motor[i] := FALSE;
        GVL.Auto_Weights[i] := 0.0;
        GVL.Auto_Target_Weights[i] := 0.0;
        PersistentVars.Ret_Actual_Weights[i] := 0.0;
        PersistentVars.Ret_Bin_Target_Weights[i] := 0.0;
    END_FOR;
    Auto_Sum_Act_Weight := 0.0;
    GVL.Auto_Total_Actual_Weight := 0.0;
    Sequence_Complete := FALSE;
    GVL.Auto_Sequence_Complete := FALSE;
    Active_Material_ID := 0;
    Active_Bin_ID := 0;
    Active_Target_Weight := 0.0;
    Active_Live_Weight := 0.0;
    GVL.Auto_Active_Target_Weight := 0.0;
    GVL.Auto_Active_Live_Weight := 0.0;
    GVL.Auto_Active_Mat := 0;
    GVL.Auto_Active_Bin := 0;
    Excess_Alarm := FALSE;
    Auto_Error_Code := 0;
    GVL.Error_Code := 0;
    Error := FALSE;
    GVL.Current_Batch_Cycle := 0;
    GVL.Completed_Batch_Cycles := 0;
    GVL.All_Cycles_Complete := FALSE;
    Auto_Completed_Batch_Cycles := 0;
    Auto_Current_Batch_Cycle := 0;
    Auto_All_Cycles_Complete := FALSE;
    GVL.Target_Batch_Cycles := 0;
    GVL.Start_Button := FALSE;
    GVL.Run := FALSE;
    Master_Run := FALSE;
    GVL.Next_Cycle_Start := FALSE;
    Next_Cycle_Ready := FALSE;
    GVL.Next_Cycle_Ready := FALSE;
    Current_Step := 0;
    Cycle_Manager_State := 0;
    Internal_FB_Start := FALSE;
    Tare_Pulse_Req := FALSE;
    Tare_Auto_Batch := FALSE;
    Waiting_Next_Batch := FALSE;
    Between_Cycle_Hold := FALSE;
    Paused_By_Hold := FALSE;
    PersistentVars.Ret_Process_Was_Active := FALSE;
    PersistentVars.Ret_Cycle_Manager_State := 0;
    PersistentVars.Ret_Current_Step := 0;
    PersistentVars.Ret_Resume_Step := 0;
    PersistentVars.Ret_bin_last_weight := 0.0;
    PersistentVars.bin_last_weight := 0.0;
    bin_last_weight := 0.0;
    Status_Message := 'Auto [Reset]: System Reset complete. Ready for Start.';
    RETURN;
END_IF;

IF Fault_Reset_Pulse THEN
    IF (Auto_Error_Code = 4) AND (load_cell_value < eff_empty_limit) AND (GVL.load_cell_auto < eff_empty_limit) THEN
        Auto_Error_Code := 0;
        GVL.Error_Code := 0;
    ELSIF (Auto_Error_Code = 10) AND (GVL.load_cell_semi_auto < eff_empty_limit) THEN
        Auto_Error_Code := 0;
        GVL.Error_Code := 0;
    ELSIF (Auto_Error_Code = 5) AND (NOT Line_Fault) THEN
        Auto_Error_Code := 0;
        GVL.Error_Code := 0;
        Paused_By_Hold := FALSE;
    ELSIF (Auto_Error_Code = 8) AND (NOT Partner_Line_Fault) THEN
        Auto_Error_Code := 0;
        GVL.Error_Code := 0;
        Paused_By_Hold := FALSE;
    END_IF;
    Error := (Auto_Error_Code > 0);
END_IF;

// Process HOLD on Safety / Fault conditions
IF NOT E_Stop_Active OR NOT Auto_Mode_DI OR (Auto_Error_Code > 0) THEN
    Paused_By_Hold := TRUE;
    FOR i := 1 TO 6 DO
        Auto_Bin[i] := FALSE;
        auto_motor_slow_trigger[i] := FALSE;
        auto_bin_motor[i] := FALSE;
        GVL.Auto_Bin[i] := FALSE;
        GVL.auto_motor_slow_trigger[i] := FALSE;
        GVL.auto_bin_motor[i] := FALSE;
    END_FOR;
ELSE
    Paused_By_Hold := FALSE;
END_IF;

// -----------------------------------------------------------------------------
// 4. MASTER CYCLE MANAGER STATE MACHINE
// -----------------------------------------------------------------------------
CASE Cycle_Manager_State OF
    0: // IDLE
        Internal_FB_Start := FALSE;
        Master_Run := FALSE;
        IF NOT PersistentVars.Ret_Process_Was_Active THEN
            GVL.Run := FALSE;
        END_IF;
        GVL.Next_Cycle_Start := FALSE;
        Next_Cycle_Ready := FALSE;
        GVL.Next_Cycle_Ready := FALSE;
        Sequence_Complete := FALSE;
        GVL.Auto_Sequence_Complete := FALSE;
        Current_Step := 0;
        GVL.Auto_Current_Step := 0;

        IF Start_Pulse THEN
            IF Target_Batch_Cycles > 0 THEN
                GVL.Target_Batch_Cycles := Target_Batch_Cycles;
            ELSIF GVL.Target_Batch_Cycles <= 0 THEN
                GVL.Target_Batch_Cycles := 1;
            END_IF;

            IF NOT E_Stop_Active THEN
                Status_Message := 'Auto [State 0]: Cannot Start - E-Stop Open!';
            ELSIF Auto_Error_Code > 0 AND Auto_Error_Code <> 4 AND Auto_Error_Code <> 10 THEN
                Status_Message := CONCAT('Auto [State 0]: Cannot Start - Error ', INT_TO_STRING(Auto_Error_Code));
            ELSIF (load_cell_value >= eff_empty_limit) OR (GVL.load_cell_auto >= eff_empty_limit) THEN
                Auto_Error_Code := 4;
                GVL.Error_Code := 4;
                Status_Message := CONCAT('Auto [State 0]: Error 4 - Auto Scale 1 not empty (< ', CONCAT(REAL_TO_STRING(eff_empty_limit), ' kg)'));
            ELSIF GVL.load_cell_semi_auto >= eff_empty_limit THEN
                Auto_Error_Code := 10;
                GVL.Error_Code := 10;
                Status_Message := CONCAT('Auto [State 0]: Error 10 - Semi Scale 2 not empty (< ', CONCAT(REAL_TO_STRING(eff_empty_limit), ' kg)'));
            ELSE
                Auto_Error_Code := 0;
                GVL.Error_Code := 0;
                GVL.Current_Batch_Cycle := 1;
                GVL.Completed_Batch_Cycles := 0;
                GVL.All_Cycles_Complete := FALSE;
                Auto_Completed_Batch_Cycles := 0;
                Auto_Current_Batch_Cycle := 1;
                Auto_All_Cycles_Complete := FALSE;
                
                // Continuous Run Active
                GVL.Run := TRUE;
                Master_Run := TRUE;
                Internal_FB_Start := TRUE;
                Cycle_Manager_State := 1;
                Current_Step := 0;
                
                bin_last_weight := 0.0;
                PersistentVars.bin_last_weight := 0.0;
                PersistentVars.Ret_bin_last_weight := 0.0;
                FOR i := 1 TO 6 DO
                    Actual_Weights[i] := 0.0;
                    PersistentVars.Ret_Actual_Weights[i] := 0.0;
                END_FOR;
                
                Tare_Pulse_Req := TRUE;
                GVL.Start_Button := FALSE;
            END_IF;
        END_IF;

    1: // RUNNING ACTIVE BATCH CYCLE
        Internal_FB_Start := TRUE;
        GVL.Run := TRUE;
        Master_Run := TRUE;
        GVL.Next_Cycle_Start := FALSE;
        Next_Cycle_Ready := FALSE;
        GVL.Next_Cycle_Ready := FALSE;

        // Dual-Sequence Completion Handshake: BOTH Auto and Semi must finish
        IF Sequence_Complete AND Semi_Sequence_Done AND (Auto_Has_Active_Bins OR Semi_Has_Active_Bins) THEN
            GVL.Completed_Batch_Cycles := GVL.Current_Batch_Cycle;
            Auto_Completed_Batch_Cycles := GVL.Current_Batch_Cycle;
            
            IF (GVL.Current_Batch_Cycle < GVL.Target_Batch_Cycles) AND (GVL.Error_Code = 0) THEN
                Internal_FB_Start := FALSE;
                Cycle_Manager_State := 5; // Transition to Between-Cycle Hold (Discharge)
                Between_Cycle_Hold := TRUE;
                // GVL.Run remains TRUE continuously throughout State 5
                Status_Message := 'Auto [Cycle Done]: Discharging hoppers - waiting for empty scale';
            ELSE
                Cycle_Manager_State := 4; // All Target Cycles Completed
                Between_Cycle_Hold := FALSE;
                GVL.Start_Button := FALSE;
            END_IF;
        END_IF;

    5: // PAUSED BETWEEN CYCLES (DISCHARGE & NEXT CYCLE READY HANDSHAKE)
        Internal_FB_Start := FALSE;
        GVL.Run := TRUE; // REMAINS TRUE until All_Cycles_Complete
        Master_Run := TRUE;
        
        // 1-Second Debounce filter for empty scale check
        IF (load_cell_value <= eff_empty_limit) AND (GVL.load_cell_auto <= eff_empty_limit) AND (GVL.load_cell_semi_auto <= eff_empty_limit) THEN
            Empty_Debounce_Timer(IN := TRUE, PT := T#1S);
            IF Empty_Debounce_Timer.Q THEN
                Next_Cycle_Ready := TRUE;
                GVL.Next_Cycle_Ready := TRUE;
                Status_Message := 'Auto [State 5]: Hoppers Empty - Ready for Next Cycle Start';
            END_IF;
        ELSE
            Empty_Debounce_Timer(IN := FALSE);
            Next_Cycle_Ready := FALSE;
            GVL.Next_Cycle_Ready := FALSE;
            Status_Message := CONCAT('Auto [State 5]: Discharging batch (Scale > ', CONCAT(REAL_TO_STRING(eff_empty_limit), ' kg)...'));
        END_IF;

        // Next Cycle Trigger Pulse
        IF Next_Cycle_Rising THEN
            IF Auto_Error_Code > 0 THEN
                Status_Message := CONCAT('Auto [State 5]: Blocked by Auto_Error_Code ', INT_TO_STRING(Auto_Error_Code));
            ELSIF Next_Cycle_Ready AND (GVL.Current_Batch_Cycle < GVL.Target_Batch_Cycles) THEN
                Next_Cycle_Ready := FALSE;
                GVL.Next_Cycle_Ready := FALSE;
                GVL.Next_Cycle_Start := FALSE;
                Next_Cycle_Last := FALSE;
                
                GVL.Current_Batch_Cycle := GVL.Current_Batch_Cycle + 1;
                Auto_Current_Batch_Cycle := GVL.Current_Batch_Cycle;
                
                Sequence_Complete := FALSE;
                GVL.Auto_Sequence_Complete := FALSE;
                GVL.Semi_Auto_Sequence_Complete := FALSE;
                Between_Cycle_Hold := FALSE;
                Cycle_Manager_State := 1;
                Current_Step := 0;
                Internal_FB_Start := TRUE;
                
                bin_last_weight := 0.0;
                PersistentVars.bin_last_weight := 0.0;
                PersistentVars.Ret_bin_last_weight := 0.0;
                FOR i := 1 TO 6 DO
                    Actual_Weights[i] := 0.0;
                    PersistentVars.Ret_Actual_Weights[i] := 0.0;
                    Auto_Bin[i] := FALSE;
                    auto_motor_slow_trigger[i] := FALSE;
                    auto_bin_motor[i] := FALSE;
                END_FOR;
                
                Tare_Pulse_Req := TRUE;
                Status_Message := CONCAT('Auto [State 5]: Cycle ', CONCAT(INT_TO_STRING(GVL.Current_Batch_Cycle), ' Started'));
            ELSE
                Status_Message := CONCAT('Auto [State 5]: Empty scale < ', CONCAT(REAL_TO_STRING(eff_empty_limit), ' kg before pressing Next Cycle!'));
            END_IF;
        END_IF;

    4: // ALL TARGET BATCH CYCLES COMPLETE
        Internal_FB_Start := FALSE;
        Between_Cycle_Hold := FALSE;
        GVL.Run := FALSE; // Turn off GVL.Run only when all cycles finish
        Master_Run := FALSE;
        GVL.Start_Button := FALSE;
        Auto_All_Cycles_Complete := TRUE;
        GVL.All_Cycles_Complete := TRUE;
        Sequence_Complete := TRUE;
        GVL.Auto_Sequence_Complete := TRUE;
        Next_Cycle_Ready := FALSE;
        GVL.Next_Cycle_Ready := FALSE;
        Status_Message := CONCAT('Auto [Finished]: All ', CONCAT(INT_TO_STRING(GVL.Target_Batch_Cycles), ' Batch Cycles Complete'));

        IF Start_Pulse THEN
            IF Scale_Empty_OK THEN
                Current_Step := 0;
                Cycle_Manager_State := 0;
                Auto_All_Cycles_Complete := FALSE;
                GVL.All_Cycles_Complete := FALSE;
            ELSE
                Auto_Error_Code := 4;
                GVL.Error_Code := 4;
                Status_Message := 'Auto [Finished]: Empty hopper before starting new job!';
            END_IF;
        END_IF;
END_CASE;

// -----------------------------------------------------------------------------
// 5. AUTO DOSING SEQUENCE (STEPS 1..6, SETTLE 7, COMPLETE 8)
// -----------------------------------------------------------------------------
IF (Current_Step = 0) AND Internal_FB_Start AND (Cycle_Manager_State = 1) THEN
    IF NOT Auto_Has_Active_Bins THEN
        Current_Step := 8;
        Sequence_Complete := TRUE;
        GVL.Auto_Sequence_Complete := TRUE;
    ELSE
        Current_Step := 1;
        bin_last_weight := load_cell_value;
        PersistentVars.Ret_bin_last_weight := bin_last_weight;
        PersistentVars.bin_last_weight := bin_last_weight;
        Last_Dosing_Step := 1;
        Sequence_Complete := FALSE;
        GVL.Auto_Sequence_Complete := FALSE;
    END_IF;
END_IF;

CASE Current_Step OF
    0:
        Active_Material_ID := 0;
        Active_Bin_ID := 0;
        Active_Target_Weight := 0.0;
        Active_Live_Weight := 0.0;
        FOR i := 1 TO 6 DO
            Auto_Bin[i] := FALSE;
            auto_motor_slow_trigger[i] := FALSE;
            auto_bin_motor[i] := FALSE;
        END_FOR;

    1..6:
        WHILE (Current_Step >= 1) AND (Current_Step <= 6) DO
            Mat_Idx := Auto_Bin_Material_Mapping[Current_Step];
            IF (Mat_Idx < 1) OR (Mat_Idx > 20) THEN
                Mat_Idx := GVL.Auto_Bin_Material_Mapping[Current_Step];
            END_IF;
            target_weight := 0.0;
            IF (Mat_Idx >= 1) AND (Mat_Idx <= 20) THEN
                target_weight := GVL.Recipe_Weights[Mat_Idx];
            END_IF;

            IF (Mat_Idx < 1) OR (Mat_Idx > 20) OR (target_weight <= 0.0) THEN
                Auto_Bin[Current_Step] := FALSE;
                auto_motor_slow_trigger[Current_Step] := FALSE;
                auto_bin_motor[Current_Step] := FALSE;
                Actual_Weights[Current_Step] := 0.0;
                IF Current_Step = 6 THEN
                    Current_Step := 7;
                    EXIT;
                ELSE
                    Current_Step := Current_Step + 1;
                END_IF;
            ELSE
                EXIT;
            END_IF;
        END_WHILE;

        IF Inter_Bin_Settling THEN
            Active_Material_ID := Settle_Hold_Mat;
            Active_Bin_ID := Settle_Hold_Step;
            Active_Target_Weight := Settle_Hold_Target;
            
            min_tol_weight := Settle_Hold_Target - Auto_Bin_Tolerance[Settle_Hold_Step];
            max_tol_weight := Settle_Hold_Target + Auto_Bin_Tolerance[Settle_Hold_Step];

            actual_bin := load_cell_value - bin_last_weight;
            IF actual_bin < 0.0 THEN
                actual_bin := 0.0;
            END_IF;
            Actual_Weights[Settle_Hold_Step] := actual_bin;
            Active_Live_Weight := actual_bin;

            CASE Inter_Bin_Settle_Arm OF
                0: // Arm settling timer
                    FOR i := 1 TO 6 DO
                        Auto_Bin[i] := FALSE;
                        auto_motor_slow_trigger[i] := FALSE;
                        auto_bin_motor[i] := FALSE;
                    END_FOR;
                    Inter_Bin_Timer(IN := FALSE);
                    Periodic_Check_Timer(IN := FALSE);
                    Inter_Bin_Settle_Arm := 1;
                    Status_Message := CONCAT('Auto [Step ', CONCAT(INT_TO_STRING(Settle_Hold_Step), ']: Settling in progress...'));

                1: // Settling delay timer running (Effective_Delay)
                    FOR i := 1 TO 6 DO
                        Auto_Bin[i] := FALSE;
                        auto_motor_slow_trigger[i] := FALSE;
                        auto_bin_motor[i] := FALSE;
                    END_FOR;
                    Inter_Bin_Timer(IN := TRUE, PT := Effective_Delay);
                    IF Inter_Bin_Timer.Q THEN
                        Inter_Bin_Timer(IN := FALSE);
                        
                        // Post-settle check
                        IF actual_bin > max_tol_weight THEN
                            IF Excess_Allowed THEN
                                // Excess allowed: lock weight and advance
                                Excess_Alarm := FALSE;
                                bin_last_weight := load_cell_value;
                                PersistentVars.Ret_bin_last_weight := bin_last_weight;
                                PersistentVars.bin_last_weight := bin_last_weight;
                                Current_Step := Inter_Bin_Next_Step;
                                Last_Dosing_Step := Current_Step;
                                Inter_Bin_Settling := FALSE;
                                Inter_Bin_Settle_Arm := 0;
                            ELSE
                                // Overfilled: trigger alarm and enter 500ms monitoring
                                Excess_Alarm := TRUE;
                                Inter_Bin_Settle_Arm := 2;
                                Periodic_Check_Timer(IN := FALSE);
                                Status_Message := CONCAT('Auto [Step ', CONCAT(INT_TO_STRING(Settle_Hold_Step), ']: Settled Overfill Alarm!'));
                            END_IF;
                        ELSIF actual_bin < min_tol_weight THEN
                            // Underfilled: enter 500ms top-up monitoring
                            Excess_Alarm := FALSE;
                            Inter_Bin_Settle_Arm := 3;
                            Periodic_Check_Timer(IN := FALSE);
                            Status_Message := CONCAT('Auto [Step ', CONCAT(INT_TO_STRING(Settle_Hold_Step), ']: Settled below Tol — Topping up'));
                        ELSE
                            // Within tolerance: lock weight and advance
                            Excess_Alarm := FALSE;
                            bin_last_weight := load_cell_value;
                            PersistentVars.Ret_bin_last_weight := bin_last_weight;
                            PersistentVars.bin_last_weight := bin_last_weight;
                            Current_Step := Inter_Bin_Next_Step;
                            Last_Dosing_Step := Current_Step;
                            Inter_Bin_Settling := FALSE;
                            Inter_Bin_Settle_Arm := 0;
                        END_IF;
                    END_IF;

                2: // State 2: Overweight 500ms periodic monitoring
                    FOR i := 1 TO 6 DO
                        Auto_Bin[i] := FALSE;
                        auto_motor_slow_trigger[i] := FALSE;
                        auto_bin_motor[i] := FALSE;
                    END_FOR;
                    
                    Periodic_Check_Timer(IN := NOT Periodic_Check_Timer.Q, PT := T#500MS);
                    IF Periodic_Check_Timer.Q THEN
                        IF Excess_Allowed OR (actual_bin <= max_tol_weight) THEN
                            // Weight back in range or excess allowed -> clear alarm and restart settling delay!
                            Excess_Alarm := FALSE;
                            Inter_Bin_Settle_Arm := 0;
                        ELSE
                            Excess_Alarm := TRUE;
                            Status_Message := CONCAT('Auto [Step ', CONCAT(INT_TO_STRING(Settle_Hold_Step), ']: Overfill! Waiting in-range / Excess'));
                        END_IF;
                    END_IF;

                3: // State 3: Underweight 500ms periodic fine top-up monitoring
                    Periodic_Check_Timer(IN := NOT Periodic_Check_Timer.Q, PT := T#500MS);
                    
                    IF (NOT Paused_By_Hold) AND GVL.Run AND (Auto_Error_Code = 0) THEN
                        IF actual_bin < min_tol_weight THEN
                            Auto_Bin[Settle_Hold_Step] := FALSE;
                            auto_motor_slow_trigger[Settle_Hold_Step] := TRUE;
                            auto_bin_motor[Settle_Hold_Step] := TRUE;
                            Status_Message := CONCAT('Auto [Step ', CONCAT(INT_TO_STRING(Settle_Hold_Step), ']: Fine Top-up in progress'));
                        ELSE
                            // Reached target range -> shut off feeders and restart settling delay!
                            Auto_Bin[Settle_Hold_Step] := FALSE;
                            auto_motor_slow_trigger[Settle_Hold_Step] := FALSE;
                            auto_bin_motor[Settle_Hold_Step] := FALSE;
                            Inter_Bin_Settle_Arm := 0;
                        END_IF;
                    ELSE
                        Auto_Bin[Settle_Hold_Step] := FALSE;
                        auto_motor_slow_trigger[Settle_Hold_Step] := FALSE;
                        auto_bin_motor[Settle_Hold_Step] := FALSE;
                    END_IF;
            END_CASE;

        ELSIF (Current_Step >= 1) AND (Current_Step <= 6) THEN
            Mat_Idx := Auto_Bin_Material_Mapping[Current_Step];
            IF (Mat_Idx < 1) OR (Mat_Idx > 20) THEN
                Mat_Idx := GVL.Auto_Bin_Material_Mapping[Current_Step];
            END_IF;
            target_weight := GVL.Recipe_Weights[Mat_Idx];
            
            IF Current_Step <> Last_Dosing_Step THEN
                bin_last_weight := load_cell_value;
                PersistentVars.Ret_bin_last_weight := bin_last_weight;
                PersistentVars.bin_last_weight := bin_last_weight;
                Last_Dosing_Step := Current_Step;
            END_IF;

            cutoff_trigger_weight := target_weight - Auto_Coarse_To_Fine_Speed[Current_Step];
            min_tol_weight := target_weight - Auto_Bin_Tolerance[Current_Step];
            max_tol_weight := target_weight + Auto_Bin_Tolerance[Current_Step];

            actual_bin := load_cell_value - bin_last_weight;
            IF actual_bin < 0.0 THEN
                actual_bin := 0.0;
            END_IF;

            Active_Material_ID := Mat_Idx;
            Active_Bin_ID := Current_Step;
            Active_Target_Weight := target_weight;

            // Continually track live weight during both Run and Safety Hold (captures extra power-off dump)
            Actual_Weights[Current_Step] := actual_bin;
            Active_Live_Weight := actual_bin;

            IF (NOT Paused_By_Hold) AND GVL.Run AND (Auto_Error_Code = 0) THEN
                IF actual_bin < cutoff_trigger_weight THEN
                    Auto_Bin[Current_Step] := TRUE;
                    auto_motor_slow_trigger[Current_Step] := FALSE;
                    auto_bin_motor[Current_Step] := TRUE;
                    Excess_Alarm := FALSE;
                    Status_Message := CONCAT('Auto [Step ', CONCAT(INT_TO_STRING(Current_Step), ']: Coarse Feeding'));
                ELSIF actual_bin < min_tol_weight THEN
                    Auto_Bin[Current_Step] := FALSE;
                    auto_motor_slow_trigger[Current_Step] := TRUE;
                    auto_bin_motor[Current_Step] := TRUE;
                    Excess_Alarm := FALSE;
                    Status_Message := CONCAT('Auto [Step ', CONCAT(INT_TO_STRING(Current_Step), ']: Fine Feeding'));
                ELSIF actual_bin > max_tol_weight THEN
                    Auto_Bin[Current_Step] := FALSE;
                    auto_motor_slow_trigger[Current_Step] := FALSE;
                    auto_bin_motor[Current_Step] := FALSE;
                    IF Excess_Allowed THEN
                        Excess_Alarm := FALSE;
                        Status_Message := CONCAT('Auto [Step ', CONCAT(INT_TO_STRING(Current_Step), ']: Target Reached (Excess Allowed)'));
                        Settle_Hold_Step := Current_Step;
                        Settle_Hold_Mat := Mat_Idx;
                        Settle_Hold_Target := target_weight;
                        IF Current_Step >= 6 THEN
                            Current_Step := 7;
                        ELSE
                            Inter_Bin_Next_Step := Current_Step + 1;
                            Inter_Bin_Settling := TRUE;
                            Inter_Bin_Settle_Arm := 0;
                        END_IF;
                    ELSE
                        Excess_Alarm := TRUE;
                        Status_Message := CONCAT('Auto [Step ', CONCAT(INT_TO_STRING(Current_Step), ']: Excess Weight Alarm!'));
                    END_IF;
                ELSE
                    Auto_Bin[Current_Step] := FALSE;
                    auto_motor_slow_trigger[Current_Step] := FALSE;
                    auto_bin_motor[Current_Step] := FALSE;
                    Excess_Alarm := FALSE;
                    Status_Message := CONCAT('Auto [Step ', CONCAT(INT_TO_STRING(Current_Step), ']: Target Reached - Advancing'));
                    Settle_Hold_Step := Current_Step;
                    Settle_Hold_Mat := Mat_Idx;
                    Settle_Hold_Target := target_weight;
                    IF Current_Step >= 6 THEN
                        Current_Step := 7;
                    ELSE
                        Inter_Bin_Next_Step := Current_Step + 1;
                        Inter_Bin_Settling := TRUE;
                        Inter_Bin_Settle_Arm := 0;
                    END_IF;
                END_IF;
            END_IF;
        END_IF;

    7: // FINAL SETTLING DELAY
        Active_Material_ID := 0;
        Active_Bin_ID := 0;
        Active_Target_Weight := 0.0;
        Active_Live_Weight := 0.0;
        FOR i := 1 TO 6 DO
            Auto_Bin[i] := FALSE;
            auto_motor_slow_trigger[i] := FALSE;
            auto_bin_motor[i] := FALSE;
        END_FOR;
        Status_Message := 'Auto [Step 7]: Settling Delay in progress...';
        Completion_Timer(IN := TRUE, PT := Effective_Delay);
        IF Completion_Timer.Q THEN
            Completion_Timer(IN := FALSE);
            Current_Step := 8;
        END_IF;

    8: // AUTO SEQUENCE COMPLETE (WAITS FOR FOLLOWER ASYNCHRONOUSLY)
        Active_Material_ID := 0;
        Active_Bin_ID := 0;
        Active_Target_Weight := 0.0;
        Active_Live_Weight := 0.0;
        FOR i := 1 TO 6 DO
            Auto_Bin[i] := FALSE;
            auto_motor_slow_trigger[i] := FALSE;
            auto_bin_motor[i] := FALSE;
        END_FOR;
        Sequence_Complete := TRUE;
        GVL.Auto_Sequence_Complete := TRUE;
        IF NOT Semi_Sequence_Done THEN
            Status_Message := 'Auto [Step 8]: Auto Finished — Waiting for Semi-Auto to complete...';
        ELSE
            Status_Message := 'Auto [Step 8]: Both Sequences Complete';
        END_IF;
END_CASE;

// -----------------------------------------------------------------------------
// 6. OUTPUT SYNCHRONIZATION & PERSISTENT SNAPSHOT
// -----------------------------------------------------------------------------
FOR i := 1 TO 6 DO
    GVL.Auto_Bin[i] := Auto_Bin[i];
    GVL.auto_motor_slow_trigger[i] := auto_motor_slow_trigger[i];
    GVL.auto_bin_motor[i] := auto_bin_motor[i];
    GVL.Auto_Weights[i] := Actual_Weights[i];
END_FOR;

Auto_Sum_Act_Weight := 0.0;
FOR i := 1 TO 6 DO
    Auto_Sum_Act_Weight := Auto_Sum_Act_Weight + Actual_Weights[i];
END_FOR;
GVL.Auto_Total_Actual_Weight := Auto_Sum_Act_Weight;

GVL.Auto_Active_Mat := Active_Material_ID;
GVL.Auto_Active_Bin := Active_Bin_ID;
GVL.Auto_Active_Target_Weight := Active_Target_Weight;
GVL.Auto_Active_Live_Weight := Active_Live_Weight;
GVL.Auto_Current_Step := Current_Step;
GVL.Auto_Excess_Alarm := Excess_Alarm;

FOR i := 1 TO 6 DO
    Mat_Idx := Auto_Bin_Material_Mapping[i];
    IF (Mat_Idx < 1) OR (Mat_Idx > 20) THEN
        Mat_Idx := GVL.Auto_Bin_Material_Mapping[i];
    END_IF;
    target_weight := 0.0;
    IF (Mat_Idx >= 1) AND (Mat_Idx <= 20) THEN
        target_weight := GVL.Recipe_Weights[Mat_Idx];
    END_IF;
    Auto_Total_Target_Set[i] := target_weight;
    GVL.Auto_Target_Weights[i] := target_weight;
END_FOR;

// Persistent Snapshot
IF Cycle_Manager_State = 4 THEN
    PersistentVars.Ret_Process_Was_Active := FALSE;
    PersistentVars.Ret_Cycle_Manager_State := 0;
    PersistentVars.Ret_Current_Step := 0;
    PersistentVars.Ret_Resume_Step := 0;
    PersistentVars.Ret_Active_Live_Weight := 0.0;
    PersistentVars.Ret_bin_last_weight := 0.0;
    FOR i := 1 TO 6 DO
        PersistentVars.Ret_Actual_Weights[i] := 0.0;
    END_FOR;
ELSIF Cycle_Manager_State = 1 OR Cycle_Manager_State = 5 THEN
    PersistentVars.Ret_Process_Was_Active := TRUE;
    PersistentVars.Ret_Cycle_Manager_State := Cycle_Manager_State;
    PersistentVars.Ret_Current_Step := Current_Step;
    IF (Current_Step >= 1) AND (Current_Step <= 6) THEN
        PersistentVars.Ret_Resume_Step := Current_Step;
    END_IF;
    PersistentVars.Ret_Current_Batch_Cycle := GVL.Current_Batch_Cycle;
    PersistentVars.Ret_Completed_Batch_Cycles := GVL.Completed_Batch_Cycles;
    PersistentVars.Ret_Target_Batch_Cycles := GVL.Target_Batch_Cycles;
    PersistentVars.Ret_Active_Material_ID := Active_Material_ID;
    PersistentVars.Ret_Active_Bin_ID := Active_Bin_ID;
    PersistentVars.Ret_Active_Target_Weight := Active_Target_Weight;
    PersistentVars.Ret_Active_Live_Weight := Active_Live_Weight;
    PersistentVars.Ret_bin_last_weight := bin_last_weight;
    FOR i := 1 TO 6 DO
        PersistentVars.Ret_Actual_Weights[i] := Actual_Weights[i];
    END_FOR;
END_IF;

// -----------------------------------------------------------------------------
// 7. TARE PULSE EMISSION (STRICT INTERLOCK)
// -----------------------------------------------------------------------------
IF Tare_Pulse_Req THEN
    IF Scale_Empty_OK AND (Cycle_Manager_State = 1) AND (Current_Step <= 1) THEN
        Tare_Auto_Batch := TRUE;
    ELSE
        Tare_Auto_Batch := FALSE;
    END_IF;
    Tare_Pulse_Req := FALSE;
ELSE
    Tare_Auto_Batch := FALSE;
END_IF;

Waiting_Next_Batch := (Cycle_Manager_State = 5) AND (GVL.Target_Batch_Cycles > 1) AND (GVL.Current_Batch_Cycle < GVL.Target_Batch_Cycles);
GVL.Waiting_Next_batch_HMI_HIDE := Waiting_Next_Batch;
Auto_Current_Batch_Cycle := GVL.Current_Batch_Cycle;
Auto_Completed_Batch_Cycles := GVL.Completed_Batch_Cycles;
Auto_All_Cycles_Complete := GVL.All_Cycles_Complete;
Partner_Semi_Current_Batch_Cycle := GVL.Current_Batch_Cycle;
Partner_Semi_Completed_Batch_Cycles := GVL.Completed_Batch_Cycles;
Partner_Semi_All_Cycles_Complete := GVL.All_Cycles_Complete;

END_FUNCTION_BLOCK

// PLC_AC500_V3/Application/Semi_Auto_Batching_V16
FUNCTION_BLOCK Semi_Auto_Batching_V16
VAR_INPUT
    Master_Run : BOOL;                                  // Master Run command from Auto_Batching_V16.Master_Run (or GVL.Run)
    Reset : BOOL;                                       // System reset pulse (clears active steps, outputs, and actual weights)
    Fault_Reset : BOOL;                                 // Rising-edge fault acknowledge
    E_Stop_Active : BOOL;                               // Emergency Stop status (NC: TRUE = Healthy, FALSE = E-Stop tripped)
    Semi_Auto_Bin_Material_Mapping : ARRAY[1..10] OF INT;// Physical Silos 1..10 to Recipe Material IDs (1..20, 0=skip)
    Semi_Auto_Bin_Tolerance : ARRAY[1..10] OF REAL;     // Allowable weight tolerance window (±kg)
    Inter_Bin_Delay : TIME := T#2S;                     // Settle delay between bins (Semi e.g. T#2S)
    Excess_Allowed : BOOL := FALSE;                     // TRUE = proceed if overfilled; FALSE = raise alarm and halt
    load_cell_value : REAL;                             // Live gross weight input from Semi-Auto scale (kg)
    Line_Fault : BOOL;                                  // Semi scale communication fault
END_VAR
VAR_OUTPUT
    Semi_Auto_Bin : ARRAY[1..10] OF BOOL;               // Bin indicator lamps / dump guidance for Silos 1..10
    Actual_Weights : ARRAY[1..10] OF REAL;              // Net material weight (kg) successfully dosed for each silo
    Semi_Auto_Sum_ActWeight : REAL;                     // Sum of Actual_Weights[1..10]
    Semi_Auto_Target_Weight : ARRAY[1..10] OF REAL;     // Per-bin target kg (bin index 1..10)
    Sequence_Complete : BOOL;                           // Handshake flag: TRUE when all mapped Semi silos complete dosing & settling
    Active_Material_ID : INT;                           // Recipe Material ID currently being dosed (1..20, 0 when idle/complete)
    Active_Bin_ID : INT;                                // Physical Silo index currently being dosed (1..10, 0 when idle/complete)
    Active_Target_Weight : REAL;                        // Target weight setpoint (kg) of active ingredient
    Active_Live_Weight : REAL;                          // Live net/tared weight (kg) of active silo
    Current_Step : INT;                                 // Real-time sequence step: 0=Idle, 1..10=Dosing, 31=Settle, 32=Complete
    Excess_Alarm : BOOL;                                // Overfill alarm
    Status_Message : STRING(80);                        // Diagnostic status message
    Tare_Semi_Auto_Batch : BOOL;                        // One-scan pulse to Semi load cell indicator
    Semi_Auto_Current_Batch_Cycle : INT;                // Active batch cycle number currently processing
    Semi_Auto_Completed_Batch_Cycles : INT;             // Total number of batch cycle loops completed successfully
    Semi_Auto_All_Cycles_Complete : BOOL;               // Flag: TRUE when all Target_Batch_Cycles have finished
END_VAR
VAR
    bin_last_weight : REAL;
    actual_bin : REAL;
    target_weight : REAL;
    min_tol_weight : REAL;
    max_tol_weight : REAL;
    Paused_By_Hold : BOOL;
    Effective_Delay : TIME;
    Inter_Bin_Settling : BOOL;
    Inter_Bin_Settle_Arm : INT;
    Inter_Bin_Timer : TON;
    Periodic_Check_Timer : TON;
    Settle_Hold_Step : INT;
    Settle_Hold_Mat : INT;
    Settle_Hold_Target : REAL;
    Inter_Bin_Next_Step : INT;
    Mat_Idx : INT;
    j_Mat : INT;
    i : INT;
    j : INT;
    Completion_Timer : TON;
    eff_empty_limit : REAL;
    Scale_Empty_OK : BOOL;
    Semi_Has_Active_Bins : BOOL;
    Auto_Has_Active_Bins : BOOL;
    Duplicate_Found : BOOL;
    Duplicate_Vs_Auto : BOOL;
    Invalid_Material_Range : BOOL;
    Weight_Limit_Error : BOOL;
    Semi_Mapping_All_Zero : BOOL;
    Last_Dosing_Step : INT;
    First_Scan_Done : BOOL;
    Reset_Last : BOOL;
    Reset_Pulse : BOOL;
    Fault_Reset_Last : BOOL;
    Fault_Reset_Pulse : BOOL;
    Master_Run_Last : BOOL;
    Master_Run_Rising : BOOL;
    Effective_Run : BOOL;
    Tare_Pulse_Req : BOOL;
    Last_Batch_Cycle : INT;
END_VAR


// -----------------------------------------------------------------------------
// 0. TIMINGS, THRESHOLDS & EDGE DETECTION
// -----------------------------------------------------------------------------
Effective_Delay := Inter_Bin_Delay;
IF Effective_Delay = T#0S THEN
    Effective_Delay := T#2S;
END_IF;

eff_empty_limit := GVL.Empty_Weight_Limit;
IF eff_empty_limit <= 0.0 THEN
    eff_empty_limit := 0.5;
END_IF;

Scale_Empty_OK := (load_cell_value < eff_empty_limit) AND (GVL.load_cell_semi_auto < eff_empty_limit);

Reset_Pulse := (Reset OR GVL.Reset) AND NOT Reset_Last;
Reset_Last := (Reset OR GVL.Reset);

Fault_Reset_Pulse := Fault_Reset AND NOT Fault_Reset_Last;
Fault_Reset_Last := Fault_Reset;

// Follow Master Run signal (fallback to GVL.Run if pin not connected)
Effective_Run := Master_Run OR GVL.Run;
Master_Run_Rising := Effective_Run AND NOT Master_Run_Last;
Master_Run_Last := Effective_Run;

// -----------------------------------------------------------------------------
// 1. FIRST SCAN POWER-RESUME & RETAIN RESTORE
// -----------------------------------------------------------------------------
IF NOT First_Scan_Done THEN
    First_Scan_Done := TRUE;
    
    // Restore Mapping Retain if GVL uninitialized
    FOR i := 1 TO 10 DO
        IF (GVL.Semi_Auto_Bin_Material_Mapping[i] = 0) AND (PersistentVars.Ret_Semi_Bin_Material_Mapping[i] > 0) THEN
            GVL.Semi_Auto_Bin_Material_Mapping[i] := PersistentVars.Ret_Semi_Bin_Material_Mapping[i];
        END_IF;
    END_FOR;

    // Power Resume: restore exact state without live load cell overwrite
    IF PersistentVars.Ret_Semi_Process_Was_Active AND (PersistentVars.Ret_Semi_Resume_Step >= 1) AND (PersistentVars.Ret_Semi_Resume_Step <= 10) THEN
        Current_Step := PersistentVars.Ret_Semi_Resume_Step;
        Last_Dosing_Step := Current_Step;

        bin_last_weight := PersistentVars.Ret_Semi_bin_last_weight;

        // Reconcile with live load cell weight to account for extra material dumped while power was off
        IF (load_cell_value >= bin_last_weight) AND NOT Line_Fault THEN
            Active_Live_Weight := load_cell_value - bin_last_weight;
            Actual_Weights[Current_Step] := Active_Live_Weight;
        ELSE
            Active_Live_Weight := PersistentVars.Ret_Semi_Active_Live_Weight;
            Actual_Weights[Current_Step] := Active_Live_Weight;
        END_IF;

        Semi_Auto_Sum_ActWeight := 0.0;
        FOR i := 1 TO 10 DO
            IF i <> Current_Step THEN
                Actual_Weights[i] := PersistentVars.Ret_Semi_Actual_Weights[i];
            END_IF;
            GVL.Semi_Auto_Weights[i] := Actual_Weights[i];
            Semi_Auto_Sum_ActWeight := Semi_Auto_Sum_ActWeight + Actual_Weights[i];
        END_FOR;
        GVL.Semi_Auto_Total_Actual_Weight := Semi_Auto_Sum_ActWeight;

        GVL.Semi_Auto_Active_Live_Weight := Active_Live_Weight;
        Active_Material_ID := PersistentVars.Ret_Semi_Active_Material_ID;
        Active_Bin_ID := PersistentVars.Ret_Semi_Active_Bin_ID;
        Active_Target_Weight := PersistentVars.Ret_Semi_Active_Target_Weight;
        GVL.Semi_Auto_Active_Mat := Active_Material_ID;
        GVL.Semi_Auto_Active_Bin := Active_Bin_ID;
        GVL.Semi_Auto_Active_Target_Weight := Active_Target_Weight;

        Paused_By_Hold := TRUE;
        Tare_Semi_Auto_Batch := FALSE;

        // Check if manual dump during power-off has already reached or exceeded target weight
        IF (Active_Target_Weight > 0.0) AND (Active_Live_Weight >= (Active_Target_Weight - Semi_Auto_Bin_Tolerance[Current_Step])) THEN
            IF Active_Live_Weight > (Active_Target_Weight + Semi_Auto_Bin_Tolerance[Current_Step]) THEN
                Status_Message := CONCAT('Semi-Auto [POWER RESUME]: Step ', CONCAT(INT_TO_STRING(Current_Step), ' Overfilled — Waiting Resume'));
            ELSE
                Status_Message := CONCAT('Semi-Auto [POWER RESUME]: Step ', CONCAT(INT_TO_STRING(Current_Step), ' Target Reached — Advancing on Resume'));
            END_IF;
        ELSE
            Status_Message := CONCAT('Semi-Auto [POWER RESUME]: Step ', CONCAT(INT_TO_STRING(Current_Step), ' Resumed — Ready to Feed'));
        END_IF;

    ELSIF PersistentVars.Ret_Semi_Current_Step = 32 THEN
        Current_Step := 32;
        Sequence_Complete := TRUE;
        GVL.Semi_Auto_Sequence_Complete := TRUE;
        FOR i := 1 TO 10 DO
            Actual_Weights[i] := PersistentVars.Ret_Semi_Actual_Weights[i];
            GVL.Semi_Auto_Weights[i] := Actual_Weights[i];
        END_FOR;
        Tare_Semi_Auto_Batch := FALSE;
        Status_Message := 'Semi-Auto [POWER RESUME]: Complete — Waiting for Next Cycle';

    ELSE
        Current_Step := 0;
        Sequence_Complete := FALSE;
        Tare_Semi_Auto_Batch := FALSE;
        Status_Message := 'Semi-Auto [Idle]: Ready — Waiting for Master Start';
    END_IF;
    Last_Batch_Cycle := PersistentVars.Ret_Semi_Last_Batch_Cycle;
END_IF;

// Retain snapshot of mappings
FOR i := 1 TO 10 DO
    PersistentVars.Ret_Semi_Bin_Material_Mapping[i] := GVL.Semi_Auto_Bin_Material_Mapping[i];
END_FOR;

// -----------------------------------------------------------------------------
// 2. CONFIGURATION CHECKS & ERROR DIAGNOSTICS
// -----------------------------------------------------------------------------
Duplicate_Found := FALSE;
Duplicate_Vs_Auto := FALSE;
Semi_Mapping_All_Zero := TRUE;
Invalid_Material_Range := FALSE;
Weight_Limit_Error := FALSE;
Semi_Has_Active_Bins := FALSE;
Auto_Has_Active_Bins := FALSE;

GVL.Semi_Auto_Total_Target_Weight := 0.0;
GVL.Semi_Auto_Material_Count := 0;

FOR i := 1 TO 10 DO
    Mat_Idx := Semi_Auto_Bin_Material_Mapping[i];
    IF (Mat_Idx < 1) OR (Mat_Idx > 20) THEN
        Mat_Idx := GVL.Semi_Auto_Bin_Material_Mapping[i];
    END_IF;
    IF Mat_Idx <> 0 THEN
        Semi_Mapping_All_Zero := FALSE;
    END_IF;
    IF (Mat_Idx < 0) OR (Mat_Idx > 20) THEN
        Invalid_Material_Range := TRUE;
    END_IF;
    IF (Mat_Idx >= 1) AND (Mat_Idx <= 20) THEN
        FOR j := 1 TO 10 DO
            IF j <> i THEN
                j_Mat := Semi_Auto_Bin_Material_Mapping[j];
                IF (j_Mat < 1) OR (j_Mat > 20) THEN
                    j_Mat := GVL.Semi_Auto_Bin_Material_Mapping[j];
                END_IF;
                IF (j_Mat = Mat_Idx) THEN
                    Duplicate_Found := TRUE;
                END_IF;
            END_IF;
        END_FOR;
        FOR j := 1 TO 6 DO
            j_Mat := GVL.Auto_Bin_Material_Mapping[j];
            IF (j_Mat = Mat_Idx) THEN
                Duplicate_Vs_Auto := TRUE;
            END_IF;
        END_FOR;
        target_weight := GVL.Recipe_Weights[Mat_Idx];
        IF target_weight > 0.0 THEN
            GVL.Semi_Auto_Total_Target_Weight := GVL.Semi_Auto_Total_Target_Weight + target_weight;
            GVL.Semi_Auto_Material_Count := GVL.Semi_Auto_Material_Count + 1;
            Semi_Has_Active_Bins := TRUE;
            IF target_weight < Semi_Auto_Bin_Tolerance[i] THEN
                Weight_Limit_Error := TRUE;
            END_IF;
        END_IF;
    END_IF;
END_FOR;

FOR i := 1 TO 6 DO
    Mat_Idx := GVL.Auto_Bin_Material_Mapping[i];
    IF (Mat_Idx >= 1) AND (Mat_Idx <= 20) THEN
        IF GVL.Recipe_Weights[Mat_Idx] > 0.0 THEN
            Auto_Has_Active_Bins := TRUE;
        END_IF;
    END_IF;
END_FOR;

// -----------------------------------------------------------------------------
// 3. MASTER RESET & FAULT RESET
// -----------------------------------------------------------------------------
IF Reset_Pulse THEN
    FOR i := 1 TO 10 DO
        Semi_Auto_Bin[i] := FALSE;
        Actual_Weights[i] := 0.0;
        Semi_Auto_Target_Weight[i] := 0.0;
        GVL.Semi_Auto_Bin[i] := FALSE;
        GVL.Semi_Auto_Weights[i] := 0.0;
        GVL.Semi_Auto_Target_Weights[i] := 0.0;
        PersistentVars.Ret_Semi_Actual_Weights[i] := 0.0;
        PersistentVars.Ret_Semi_Bin_Target_Weights[i] := 0.0;
    END_FOR;
    Semi_Auto_Sum_ActWeight := 0.0;
    GVL.Semi_Auto_Total_Actual_Weight := 0.0;
    Sequence_Complete := FALSE;
    GVL.Semi_Auto_Sequence_Complete := FALSE;
    Active_Material_ID := 0;
    Active_Bin_ID := 0;
    Active_Target_Weight := 0.0;
    Active_Live_Weight := 0.0;
    GVL.Semi_Auto_Active_Target_Weight := 0.0;
    GVL.Semi_Auto_Active_Live_Weight := 0.0;
    GVL.Semi_Auto_Active_Mat := 0;
    GVL.Semi_Auto_Active_Bin := 0;
    Excess_Alarm := FALSE;
    Inter_Bin_Settling := FALSE;
    Inter_Bin_Settle_Arm := 0;
    Current_Step := 0;
    Tare_Semi_Auto_Batch := FALSE;
    Paused_By_Hold := FALSE;
    PersistentVars.Ret_Semi_Process_Was_Active := FALSE;
    PersistentVars.Ret_Semi_Current_Step := 0;
    PersistentVars.Ret_Semi_Resume_Step := 0;
    PersistentVars.Ret_Semi_bin_last_weight := 0.0;
    bin_last_weight := 0.0;
    Last_Batch_Cycle := 0;
    Status_Message := 'Semi-Auto [Reset]: System Reset complete.';
    RETURN;
END_IF;

IF Fault_Reset_Pulse THEN
    IF NOT Line_Fault AND (GVL.Error_Code = 0) THEN
        Paused_By_Hold := FALSE;
    END_IF;
END_IF;

// Safety & Master Error Hold
IF (NOT E_Stop_Active) OR (GVL.Error_Code > 0) OR Line_Fault THEN
    Paused_By_Hold := TRUE;
    FOR i := 1 TO 10 DO
        Semi_Auto_Bin[i] := FALSE;
        GVL.Semi_Auto_Bin[i] := FALSE;
    END_FOR;
ELSE
    Paused_By_Hold := FALSE;
END_IF;

// -----------------------------------------------------------------------------
// 4. FOLLOWER EXECUTION (CONTROLLED BY MASTER_RUN & BATCH CYCLE ADVANCEMENT)
// -----------------------------------------------------------------------------
// Trigger fresh cycle start on Master_Run rising edge OR when GVL.Current_Batch_Cycle increments
IF Master_Run_Rising 
   OR (Effective_Run AND (Current_Step = 0) AND (GVL.Current_Batch_Cycle > 0)) 
   OR (Effective_Run AND (GVL.Current_Batch_Cycle > Last_Batch_Cycle) AND (GVL.Current_Batch_Cycle > 0)) THEN

    Last_Batch_Cycle := GVL.Current_Batch_Cycle;
    IF NOT Semi_Has_Active_Bins THEN
        Current_Step := 32;
        Sequence_Complete := TRUE;
        GVL.Semi_Auto_Sequence_Complete := TRUE;
    ELSE
        Current_Step := 1;
        Last_Dosing_Step := 1;
        bin_last_weight := load_cell_value;
        PersistentVars.Ret_Semi_bin_last_weight := bin_last_weight;
        Sequence_Complete := FALSE;
        GVL.Semi_Auto_Sequence_Complete := FALSE;
        FOR i := 1 TO 10 DO
            Actual_Weights[i] := 0.0;
            PersistentVars.Ret_Semi_Actual_Weights[i] := 0.0;
        END_FOR;
        IF Scale_Empty_OK THEN
            Tare_Pulse_Req := TRUE;
        END_IF;
    END_IF;
END_IF;

// Tare pulse emission
IF Tare_Pulse_Req THEN
    IF Scale_Empty_OK AND Effective_Run AND (Current_Step <= 1) THEN
        Tare_Semi_Auto_Batch := TRUE;
    ELSE
        Tare_Semi_Auto_Batch := FALSE;
    END_IF;
    Tare_Pulse_Req := FALSE;
ELSE
    Tare_Semi_Auto_Batch := FALSE;
END_IF;

// -----------------------------------------------------------------------------
// 5. SEMI-AUTO DOSING SEQUENCE (STEPS 1..10, SETTLE 31, COMPLETE 32)
// -----------------------------------------------------------------------------
CASE Current_Step OF
    0:
        Active_Material_ID := 0;
        Active_Bin_ID := 0;
        Active_Target_Weight := 0.0;
        Active_Live_Weight := 0.0;
        FOR i := 1 TO 10 DO
            Semi_Auto_Bin[i] := FALSE;
        END_FOR;

    1..10:
        WHILE (Current_Step >= 1) AND (Current_Step <= 10) DO
            Mat_Idx := Semi_Auto_Bin_Material_Mapping[Current_Step];
            IF (Mat_Idx < 1) OR (Mat_Idx > 20) THEN
                Mat_Idx := GVL.Semi_Auto_Bin_Material_Mapping[Current_Step];
            END_IF;
            target_weight := 0.0;
            IF (Mat_Idx >= 1) AND (Mat_Idx <= 20) THEN
                target_weight := GVL.Recipe_Weights[Mat_Idx];
            END_IF;

            IF (Mat_Idx < 1) OR (Mat_Idx > 20) OR (target_weight <= 0.0) THEN
                Semi_Auto_Bin[Current_Step] := FALSE;
                Actual_Weights[Current_Step] := 0.0;
                IF Current_Step = 10 THEN
                    Current_Step := 31;
                    EXIT;
                ELSE
                    Current_Step := Current_Step + 1;
                END_IF;
            ELSE
                EXIT;
            END_IF;
        END_WHILE;

        IF Inter_Bin_Settling THEN
            Active_Material_ID := Settle_Hold_Mat;
            Active_Bin_ID := Settle_Hold_Step;
            Active_Target_Weight := Settle_Hold_Target;
            
            min_tol_weight := Settle_Hold_Target - Semi_Auto_Bin_Tolerance[Settle_Hold_Step];
            max_tol_weight := Settle_Hold_Target + Semi_Auto_Bin_Tolerance[Settle_Hold_Step];

            actual_bin := load_cell_value - bin_last_weight;
            IF actual_bin < 0.0 THEN
                actual_bin := 0.0;
            END_IF;
            Actual_Weights[Settle_Hold_Step] := actual_bin;
            Active_Live_Weight := actual_bin;

            CASE Inter_Bin_Settle_Arm OF
                0: // Arm settling timer
                    FOR i := 1 TO 10 DO
                        Semi_Auto_Bin[i] := FALSE;
                    END_FOR;
                    Inter_Bin_Timer(IN := FALSE);
                    Periodic_Check_Timer(IN := FALSE);
                    Inter_Bin_Settle_Arm := 1;
                    Status_Message := CONCAT('Semi-Auto [Step ', CONCAT(INT_TO_STRING(Settle_Hold_Step), ']: Settling in progress...'));

                1: // Settling delay timer running (Effective_Delay)
                    FOR i := 1 TO 10 DO
                        Semi_Auto_Bin[i] := FALSE;
                    END_FOR;
                    Inter_Bin_Timer(IN := TRUE, PT := Effective_Delay);
                    IF Inter_Bin_Timer.Q THEN
                        Inter_Bin_Timer(IN := FALSE);
                        
                        // Post-settle check
                        IF actual_bin > max_tol_weight THEN
                            IF Excess_Allowed THEN
                                // Excess allowed: lock weight and advance
                                Excess_Alarm := FALSE;
                                bin_last_weight := load_cell_value;
                                PersistentVars.Ret_Semi_bin_last_weight := bin_last_weight;
                                Current_Step := Inter_Bin_Next_Step;
                                Last_Dosing_Step := Current_Step;
                                Inter_Bin_Settling := FALSE;
                                Inter_Bin_Settle_Arm := 0;
                            ELSE
                                // Overfilled: trigger alarm and enter 500ms monitoring
                                Excess_Alarm := TRUE;
                                Inter_Bin_Settle_Arm := 2;
                                Periodic_Check_Timer(IN := FALSE);
                                Status_Message := CONCAT('Semi-Auto [Step ', CONCAT(INT_TO_STRING(Settle_Hold_Step), ']: Settled Overfill Alarm!'));
                            END_IF;
                        ELSIF actual_bin < min_tol_weight THEN
                            // Underfilled: enter 500ms top-up monitoring
                            Excess_Alarm := FALSE;
                            Inter_Bin_Settle_Arm := 3;
                            Periodic_Check_Timer(IN := FALSE);
                            Status_Message := CONCAT('Semi-Auto [Step ', CONCAT(INT_TO_STRING(Settle_Hold_Step), ']: Settled below Tol — Top up needed'));
                        ELSE
                            // Within tolerance: lock weight and advance
                            Excess_Alarm := FALSE;
                            bin_last_weight := load_cell_value;
                            PersistentVars.Ret_Semi_bin_last_weight := bin_last_weight;
                            Current_Step := Inter_Bin_Next_Step;
                            Last_Dosing_Step := Current_Step;
                            Inter_Bin_Settling := FALSE;
                            Inter_Bin_Settle_Arm := 0;
                        END_IF;
                    END_IF;

                2: // State 2: Overweight 500ms periodic monitoring
                    FOR i := 1 TO 10 DO
                        Semi_Auto_Bin[i] := FALSE;
                    END_FOR;
                    
                    Periodic_Check_Timer(IN := NOT Periodic_Check_Timer.Q, PT := T#500MS);
                    IF Periodic_Check_Timer.Q THEN
                        IF Excess_Allowed OR (actual_bin <= max_tol_weight) THEN
                            // Weight back in range or excess allowed -> clear alarm and restart settling delay!
                            Excess_Alarm := FALSE;
                            Inter_Bin_Settle_Arm := 0;
                        ELSE
                            Excess_Alarm := TRUE;
                            Status_Message := CONCAT('Semi-Auto [Step ', CONCAT(INT_TO_STRING(Settle_Hold_Step), ']: Overfill! Waiting in-range / Excess'));
                        END_IF;
                    END_IF;

                3: // State 3: Underweight 500ms periodic top-up monitoring
                    Periodic_Check_Timer(IN := NOT Periodic_Check_Timer.Q, PT := T#500MS);
                    
                    IF (NOT Paused_By_Hold) AND Effective_Run AND (GVL.Error_Code = 0) THEN
                        IF actual_bin < min_tol_weight THEN
                            Semi_Auto_Bin[Settle_Hold_Step] := TRUE;
                            Status_Message := CONCAT('Semi-Auto [Step ', CONCAT(INT_TO_STRING(Settle_Hold_Step), ']: Human Dumping Top-up...'));
                        ELSE
                            // Reached target range -> shut off lamp and restart settling delay!
                            Semi_Auto_Bin[Settle_Hold_Step] := FALSE;
                            Inter_Bin_Settle_Arm := 0;
                        END_IF;
                    ELSE
                        Semi_Auto_Bin[Settle_Hold_Step] := FALSE;
                    END_IF;
            END_CASE;

        ELSIF (Current_Step >= 1) AND (Current_Step <= 10) THEN
            Mat_Idx := Semi_Auto_Bin_Material_Mapping[Current_Step];
            IF (Mat_Idx < 1) OR (Mat_Idx > 20) THEN
                Mat_Idx := GVL.Semi_Auto_Bin_Material_Mapping[Current_Step];
            END_IF;
            target_weight := GVL.Recipe_Weights[Mat_Idx];
            
            IF Current_Step <> Last_Dosing_Step THEN
                bin_last_weight := load_cell_value;
                PersistentVars.Ret_Semi_bin_last_weight := bin_last_weight;
                Last_Dosing_Step := Current_Step;
            END_IF;

            min_tol_weight := target_weight - Semi_Auto_Bin_Tolerance[Current_Step];
            max_tol_weight := target_weight + Semi_Auto_Bin_Tolerance[Current_Step];

            actual_bin := load_cell_value - bin_last_weight;
            IF actual_bin < 0.0 THEN
                actual_bin := 0.0;
            END_IF;

            Active_Material_ID := Mat_Idx;
            Active_Bin_ID := Current_Step;
            Active_Target_Weight := target_weight;

            // Continually track live weight during both Run and Safety Hold (captures extra manual power-off dump)
            Actual_Weights[Current_Step] := actual_bin;
            Active_Live_Weight := actual_bin;

            IF (NOT Paused_By_Hold) AND Effective_Run AND (GVL.Error_Code = 0) THEN
                IF actual_bin < min_tol_weight THEN
                    Semi_Auto_Bin[Current_Step] := TRUE;
                    Excess_Alarm := FALSE;
                    Status_Message := CONCAT('Semi-Auto [Step ', CONCAT(INT_TO_STRING(Current_Step), ']: Human Dumping...'));
                ELSIF actual_bin > max_tol_weight THEN
                    Semi_Auto_Bin[Current_Step] := FALSE;
                    IF Excess_Allowed THEN
                        Excess_Alarm := FALSE;
                        Status_Message := CONCAT('Semi-Auto [Step ', CONCAT(INT_TO_STRING(Current_Step), ']: Target Reached (Excess Allowed)'));
                        Settle_Hold_Step := Current_Step;
                        Settle_Hold_Mat := Mat_Idx;
                        Settle_Hold_Target := target_weight;
                        IF Current_Step >= 10 THEN
                            Current_Step := 31;
                        ELSE
                            Inter_Bin_Next_Step := Current_Step + 1;
                            Inter_Bin_Settling := TRUE;
                            Inter_Bin_Settle_Arm := 0;
                        END_IF;
                    ELSE
                        Excess_Alarm := TRUE;
                        Status_Message := CONCAT('Semi-Auto [Step ', CONCAT(INT_TO_STRING(Current_Step), ']: Excess Weight Alarm!'));
                    END_IF;
                ELSE
                    Semi_Auto_Bin[Current_Step] := FALSE;
                    Excess_Alarm := FALSE;
                    Status_Message := CONCAT('Semi-Auto [Step ', CONCAT(INT_TO_STRING(Current_Step), ']: Target Reached - Advancing'));
                    Settle_Hold_Step := Current_Step;
                    Settle_Hold_Mat := Mat_Idx;
                    Settle_Hold_Target := target_weight;
                    IF Current_Step >= 10 THEN
                        Current_Step := 31;
                    ELSE
                        Inter_Bin_Next_Step := Current_Step + 1;
                        Inter_Bin_Settling := TRUE;
                        Inter_Bin_Settle_Arm := 0;
                    END_IF;
                END_IF;
            END_IF;
        END_IF;

    31: // FINAL SETTLING DELAY
        Active_Material_ID := 0;
        Active_Bin_ID := 0;
        Active_Target_Weight := 0.0;
        Active_Live_Weight := 0.0;
        FOR i := 1 TO 10 DO
            Semi_Auto_Bin[i] := FALSE;
        END_FOR;
        Status_Message := 'Semi-Auto [Step 31]: Settling Delay in progress...';
        Completion_Timer(IN := TRUE, PT := Effective_Delay);
        IF Completion_Timer.Q THEN
            Completion_Timer(IN := FALSE);
            Current_Step := 32;
        END_IF;

    32: // SEMI-AUTO SEQUENCE COMPLETE (WAITS FOR MASTER/PARTNER ASYNCHRONOUSLY)
        Active_Material_ID := 0;
        Active_Bin_ID := 0;
        Active_Target_Weight := 0.0;
        Active_Live_Weight := 0.0;
        FOR i := 1 TO 10 DO
            Semi_Auto_Bin[i] := FALSE;
        END_FOR;
        Sequence_Complete := TRUE;
        GVL.Semi_Auto_Sequence_Complete := TRUE;
        IF NOT GVL.Auto_Sequence_Complete THEN
            Status_Message := 'Semi-Auto [Step 32]: Semi Finished — Waiting for Auto to complete...';
        ELSE
            Status_Message := 'Semi-Auto [Step 32]: Both Sequences Complete';
        END_IF;
END_CASE;

// -----------------------------------------------------------------------------
// 6. OUTPUT SYNCHRONIZATION & PERSISTENT SNAPSHOT
// -----------------------------------------------------------------------------
FOR i := 1 TO 10 DO
    GVL.Semi_Auto_Bin[i] := Semi_Auto_Bin[i];
    GVL.Semi_Auto_Weights[i] := Actual_Weights[i];
END_FOR;

Semi_Auto_Sum_ActWeight := 0.0;
FOR i := 1 TO 10 DO
    Semi_Auto_Sum_ActWeight := Semi_Auto_Sum_ActWeight + Actual_Weights[i];
END_FOR;
GVL.Semi_Auto_Total_Actual_Weight := Semi_Auto_Sum_ActWeight;

GVL.Semi_Auto_Active_Mat := Active_Material_ID;
GVL.Semi_Auto_Active_Bin := Active_Bin_ID;
GVL.Semi_Auto_Active_Target_Weight := Active_Target_Weight;
GVL.Semi_Auto_Active_Live_Weight := Active_Live_Weight;
GVL.Semi_Auto_Current_Step := Current_Step;
GVL.Semi_Auto_Excess_Alarm := Excess_Alarm;

Semi_Auto_Current_Batch_Cycle := GVL.Current_Batch_Cycle;
Semi_Auto_Completed_Batch_Cycles := GVL.Completed_Batch_Cycles;
Semi_Auto_All_Cycles_Complete := GVL.All_Cycles_Complete;

FOR i := 1 TO 10 DO
    Mat_Idx := Semi_Auto_Bin_Material_Mapping[i];
    IF (Mat_Idx < 1) OR (Mat_Idx > 20) THEN
        Mat_Idx := GVL.Semi_Auto_Bin_Material_Mapping[i];
    END_IF;
    target_weight := 0.0;
    IF (Mat_Idx >= 1) AND (Mat_Idx <= 20) THEN
        target_weight := GVL.Recipe_Weights[Mat_Idx];
    END_IF;
    Semi_Auto_Target_Weight[i] := target_weight;
    GVL.Semi_Auto_Target_Weights[i] := target_weight;
END_FOR;

// Persistent Snapshot
IF NOT Effective_Run AND (Current_Step = 0 OR Current_Step = 32) THEN
    PersistentVars.Ret_Semi_Process_Was_Active := FALSE;
    PersistentVars.Ret_Semi_Current_Step := 0;
    PersistentVars.Ret_Semi_Resume_Step := 0;
    PersistentVars.Ret_Semi_Active_Live_Weight := 0.0;
    PersistentVars.Ret_Semi_bin_last_weight := 0.0;
    FOR i := 1 TO 10 DO
        PersistentVars.Ret_Semi_Actual_Weights[i] := 0.0;
    END_FOR;
ELSIF Effective_Run THEN
    PersistentVars.Ret_Semi_Process_Was_Active := TRUE;
    PersistentVars.Ret_Semi_Current_Step := Current_Step;
    IF (Current_Step >= 1) AND (Current_Step <= 10) THEN
        PersistentVars.Ret_Semi_Resume_Step := Current_Step;
    END_IF;
    PersistentVars.Ret_Semi_Active_Material_ID := Active_Material_ID;
    PersistentVars.Ret_Semi_Active_Bin_ID := Active_Bin_ID;
    PersistentVars.Ret_Semi_Active_Target_Weight := Active_Target_Weight;
    PersistentVars.Ret_Semi_Active_Live_Weight := Active_Live_Weight;
    PersistentVars.Ret_Semi_bin_last_weight := bin_last_weight;
    PersistentVars.Ret_Semi_Last_Batch_Cycle := Last_Batch_Cycle;
    FOR i := 1 TO 10 DO
        PersistentVars.Ret_Semi_Actual_Weights[i] := Actual_Weights[i];
    END_FOR;
END_IF;

END_FUNCTION_BLOCK

// PLC_AC500_V3/Application/FB_Samyak_Control
FUNCTION_BLOCK FB_Samyak_Control
VAR_INPUT
    Com_Slot      : BYTE := 1;     (* PLC COM port *)
    Slave_Dev_ID  : BYTE := 1;     (* Samyak slave ID *)
    iDivisor      : REAL := 10.0;  (* Scale factor: Weight_Scaled = Raw / iDivisor *)
    xTare_In      : BOOL;           (* Logic tare pulse *)
    xManual_Tare  : BOOL;           (* HMI/manual tare pulse *)
END_VAR

VAR_OUTPUT
    xStatus_Done   : BOOL;
    xStatus_Busy   : BOOL;
    xStatus_Error  : BOOL;
    iTotalErrCount : INT := 0;
    xLine_Fault    : BOOL;
    Weight_Raw     : DINT;
    Weight_Scaled  : REAL;
    wError_Code    : WORD; (* Check PLC & SAMYAK BaudRate, DevId, Parity; also check PLC serial port LED blink status and RS485 connection if error repeats *)
END_VAR

VAR
    fbRead         : ModRtuMast;
    fbTare         : ModRtuMast;
    iStep          : INT := 0;
    Samyak_Buffer  : ARRAY[0..17] OF WORD;
    wTareCommand   : WORD := 1;

    rtTareTrig     : R_TRIG;
    rtErrTrig      : R_TRIG;
    tStuckWatchdog : TON;
    tRecoveryTimer : TON;

    xTareReq       : BOOL := FALSE; (* Internal tare request latch *)
END_VAR


(* --- 1) Error Tracking + Auto Recovery --- *)
tStuckWatchdog(IN := (fbRead.Busy OR fbTare.Busy), PT := T#2000MS);

rtErrTrig(CLK := (fbRead.Error OR fbTare.Error));
IF rtErrTrig.Q THEN
    iTotalErrCount := iTotalErrCount + 1;
END_IF

IF fbRead.Done OR fbTare.Done THEN
    iTotalErrCount := 0;
    xLine_Fault := FALSE;
END_IF

IF iTotalErrCount >= 10 THEN
    xLine_Fault := TRUE;
END_IF

tRecoveryTimer(IN := xLine_Fault, PT := T#5S);
IF tRecoveryTimer.Q THEN
    iTotalErrCount := 0;
    xLine_Fault := FALSE;
END_IF

IF tStuckWatchdog.Q THEN
    iStep := 99;
END_IF

(* Capture tare request from either input pulse *)
rtTareTrig(CLK := xTare_In OR xManual_Tare);
IF rtTareTrig.Q THEN
    xTareReq := TRUE;
END_IF

(* --- 2) Modbus State Machine --- *)
CASE iStep OF

    0:  (* Continuous Read *)
        fbTare(Execute := FALSE);

        fbRead(
            Execute := NOT (fbRead.Done OR fbRead.Error OR fbRead.Busy)
                       AND NOT xTareReq
                       AND NOT xLine_Fault,
            COM     := Com_Slot,
            Serv    := Slave_Dev_ID,
            FCT     := 3,
            Addr    := 0,
            Nb      := 2,
            Data    := ADR(Samyak_Buffer[0]),
            Timeout := 400,
            Done    => xStatus_Done,
            Busy    => xStatus_Busy,
            Error   => xStatus_Error,
            ErrorID => wError_Code
        );

        IF xStatus_Done THEN
            Weight_Raw := TO_DINT(SHL(TO_DWORD(Samyak_Buffer[1]), 16) OR TO_DWORD(Samyak_Buffer[0]));
            Weight_Scaled := TO_REAL(Weight_Raw) / iDivisor;
        END_IF

        IF xTareReq THEN
            iStep := 1;
        END_IF

    1:  (* Port Release *)
        fbRead(Execute := FALSE);
        IF NOT fbRead.Busy THEN
            iStep := 2;
        END_IF

    2:  (* Execute Tare *)
        fbTare(
            Execute := TRUE,
            COM     := Com_Slot,
            Serv    := Slave_Dev_ID,
            FCT     := 6,
            Addr    := 16,
            Nb      := 1,
            Data    := ADR(wTareCommand),
            Timeout := 1000,
            Done    => xStatus_Done,
            Busy    => xStatus_Busy,
            Error   => xStatus_Error,
            ErrorID => wError_Code
        );

        IF fbTare.Done OR fbTare.Error THEN
            xTareReq := FALSE;
            iStep := 3;
        END_IF

    3:  (* Return to Read *)
        fbTare(Execute := FALSE);
        IF NOT fbTare.Busy THEN
            iStep := 0;
        END_IF

    99: (* Emergency Recovery *)
        fbRead(Execute := FALSE);
        fbTare(Execute := FALSE);

        IF NOT (fbRead.Busy OR fbTare.Busy) THEN
            iTotalErrCount := 0;
            iStep := 0;
        END_IF

END_CASE

END_FUNCTION_BLOCK

